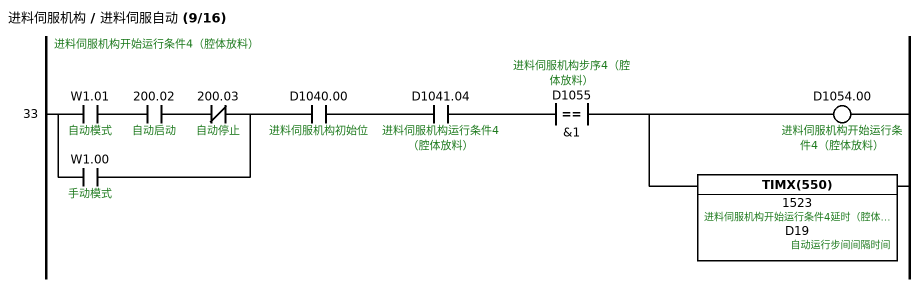
; [picture p120: 进料伺服机构 / 进料伺服自动, rungs 33-33]
; rung 33: 进料伺服机构开始运行条件4（腔体放料）
LD W1.01  ; 自动模式
AND 200.02  ; 自动启动
ANDNOT 200.03  ; 自动停止
OR W1.00  ; 手动模式
AND D1040.00  ; 进料伺服机构初始位
AND D1041.04  ; 进料伺服机构运行条件4（腔体放料）
AND=(300) D1055 &1  ; 进料伺服机构步序4（腔体放料）
OUT D1054.00  ; 进料伺服机构开始运行条件4（腔体放料）
TIMX(550) 1523 D19  ; 自动运行步间间隔时间, 进料伺服机构开始运行条件4延时（腔体放料）

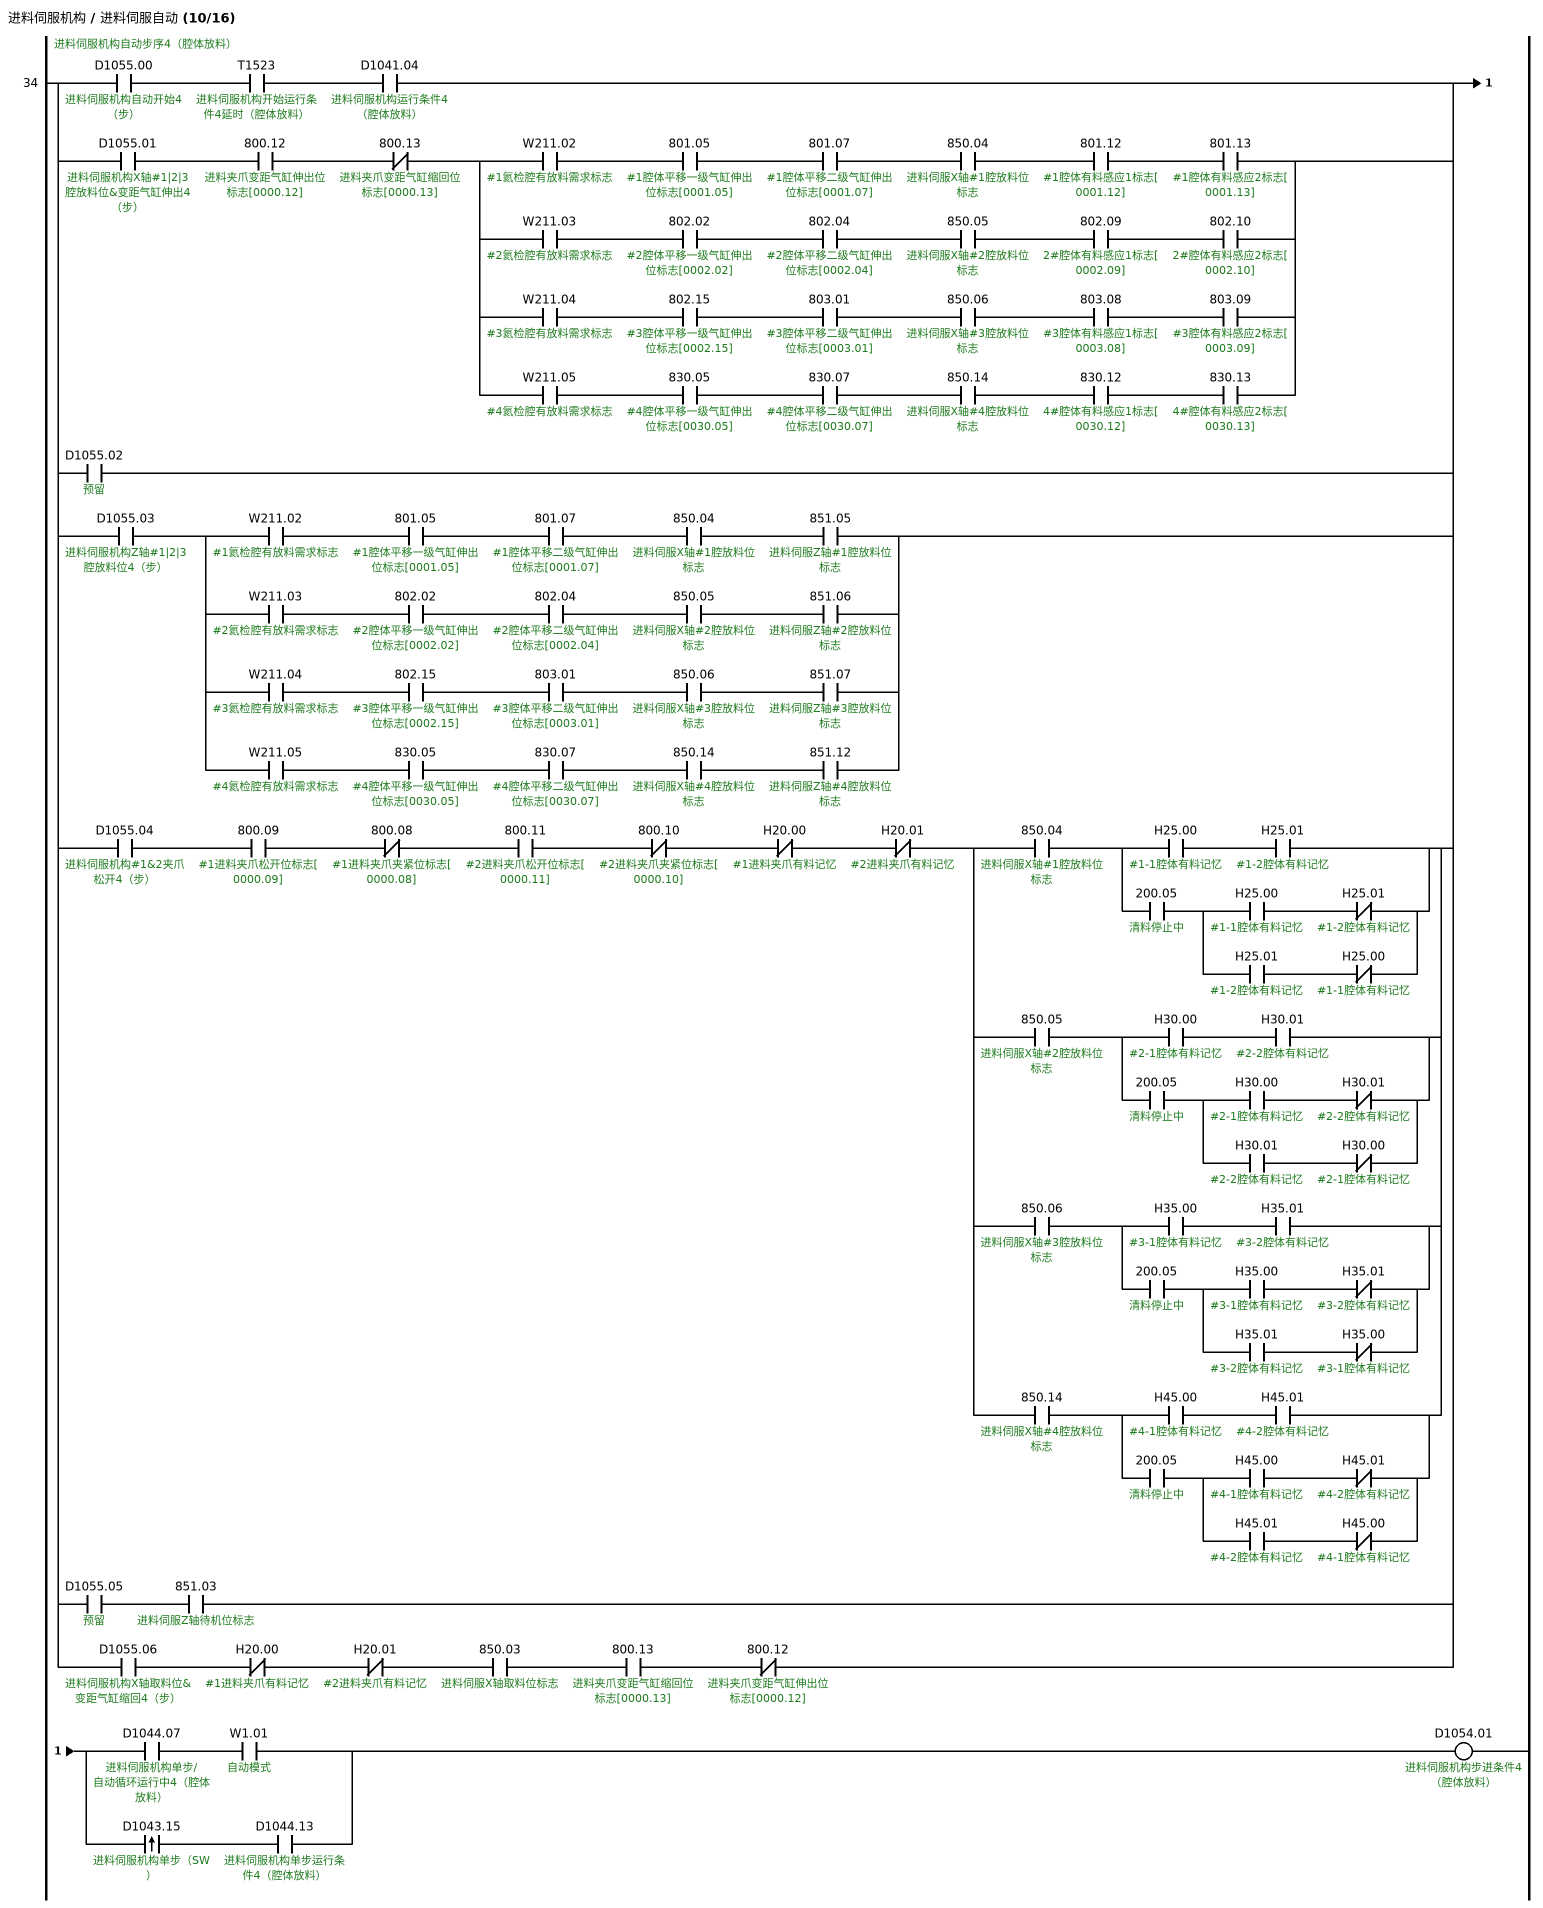
; rung 34: 进料伺服机构自动步序4（腔体放料）
LD D1055.00  ; 进料伺服机构自动开始4（步）
AND T1523  ; 进料伺服机构开始运行条件4延时（腔体放料）
AND D1041.04  ; 进料伺服机构运行条件4（腔体放料）
LD D1055.01  ; 进料伺服机构X轴#1|2|3腔放料位&变距气缸伸出4（步）
AND 800.12  ; 进料夹爪变距气缸伸出位标志[0000.12]
ANDNOT 800.13  ; 进料夹爪变距气缸缩回位标志[0000.13]
LD W211.02  ; #1氦检腔有放料需求标志
AND 801.05  ; #1腔体平移一级气缸伸出位标志[0001.05]
AND 801.07  ; #1腔体平移二级气缸伸出位标志[0001.07]
AND 850.04  ; 进料伺服X轴#1腔放料位标志
AND 801.12  ; #1腔体有料感应1标志[0001.12]
AND 801.13  ; #1腔体有料感应2标志[0001.13]
LD W211.03  ; #2氦检腔有放料需求标志
AND 802.02  ; #2腔体平移一级气缸伸出位标志[0002.02]
AND 802.04  ; #2腔体平移二级气缸伸出位标志[0002.04]
AND 850.05  ; 进料伺服X轴#2腔放料位标志
AND 802.09  ; 2#腔体有料感应1标志[0002.09]
AND 802.10  ; 2#腔体有料感应2标志[0002.10]
ORLD
LD W211.04  ; #3氦检腔有放料需求标志
AND 802.15  ; #3腔体平移一级气缸伸出位标志[0002.15]
AND 803.01  ; #3腔体平移二级气缸伸出位标志[0003.01]
AND 850.06  ; 进料伺服X轴#3腔放料位标志
AND 803.08  ; #3腔体有料感应1标志[0003.08]
AND 803.09  ; #3腔体有料感应2标志[0003.09]
ORLD
LD W211.05  ; #4氦检腔有放料需求标志
AND 830.05  ; #4腔体平移一级气缸伸出位标志[0030.05]
AND 830.07  ; #4腔体平移二级气缸伸出位标志[0030.07]
AND 850.14  ; 进料伺服X轴#4腔放料位标志
AND 830.12  ; 4#腔体有料感应1标志[0030.12]
AND 830.13  ; 4#腔体有料感应2标志[0030.13]
ORLD
ANDLD
ORLD
OR D1055.02  ; 预留
LD D1055.03  ; 进料伺服机构Z轴#1|2|3腔放料位4（步）
LD W211.02  ; #1氦检腔有放料需求标志
AND 801.05  ; #1腔体平移一级气缸伸出位标志[0001.05]
AND 801.07  ; #1腔体平移二级气缸伸出位标志[0001.07]
AND 850.04  ; 进料伺服X轴#1腔放料位标志
AND 851.05  ; 进料伺服Z轴#1腔放料位标志
LD W211.03  ; #2氦检腔有放料需求标志
AND 802.02  ; #2腔体平移一级气缸伸出位标志[0002.02]
AND 802.04  ; #2腔体平移二级气缸伸出位标志[0002.04]
AND 850.05  ; 进料伺服X轴#2腔放料位标志
AND 851.06  ; 进料伺服Z轴#2腔放料位标志
ORLD
LD W211.04  ; #3氦检腔有放料需求标志
AND 802.15  ; #3腔体平移一级气缸伸出位标志[0002.15]
AND 803.01  ; #3腔体平移二级气缸伸出位标志[0003.01]
AND 850.06  ; 进料伺服X轴#3腔放料位标志
AND 851.07  ; 进料伺服Z轴#3腔放料位标志
ORLD
LD W211.05  ; #4氦检腔有放料需求标志
AND 830.05  ; #4腔体平移一级气缸伸出位标志[0030.05]
AND 830.07  ; #4腔体平移二级气缸伸出位标志[0030.07]
AND 850.14  ; 进料伺服X轴#4腔放料位标志
AND 851.12  ; 进料伺服Z轴#4腔放料位标志
ORLD
ANDLD
ORLD
LD D1055.04  ; 进料伺服机构#1&2夹爪松开4（步）
AND 800.09  ; #1进料夹爪松开位标志[0000.09]
ANDNOT 800.08  ; #1进料夹爪夹紧位标志[0000.08]
AND 800.11  ; #2进料夹爪松开位标志[0000.11]
ANDNOT 800.10  ; #2进料夹爪夹紧位标志[0000.10]
ANDNOT H20.00  ; #1进料夹爪有料记忆
ANDNOT H20.01  ; #2进料夹爪有料记忆
LD 850.04  ; 进料伺服X轴#1腔放料位标志
LD H25.00  ; #1-1腔体有料记忆
AND H25.01  ; #1-2腔体有料记忆
LD 200.05  ; 清料停止中
LD H25.00  ; #1-1腔体有料记忆
ANDNOT H25.01  ; #1-2腔体有料记忆
LD H25.01  ; #1-2腔体有料记忆
ANDNOT H25.00  ; #1-1腔体有料记忆
ORLD
ANDLD
ORLD
ANDLD
LD 850.05  ; 进料伺服X轴#2腔放料位标志
LD H30.00  ; #2-1腔体有料记忆
AND H30.01  ; #2-2腔体有料记忆
LD 200.05  ; 清料停止中
LD H30.00  ; #2-1腔体有料记忆
ANDNOT H30.01  ; #2-2腔体有料记忆
LD H30.01  ; #2-2腔体有料记忆
ANDNOT H30.00  ; #2-1腔体有料记忆
ORLD
ANDLD
ORLD
ANDLD
ORLD
LD 850.06  ; 进料伺服X轴#3腔放料位标志
LD H35.00  ; #3-1腔体有料记忆
AND H35.01  ; #3-2腔体有料记忆
LD 200.05  ; 清料停止中
LD H35.00  ; #3-1腔体有料记忆
ANDNOT H35.01  ; #3-2腔体有料记忆
LD H35.01  ; #3-2腔体有料记忆
ANDNOT H35.00  ; #3-1腔体有料记忆
ORLD
ANDLD
ORLD
ANDLD
ORLD
LD 850.14  ; 进料伺服X轴#4腔放料位标志
LD H45.00  ; #4-1腔体有料记忆
AND H45.01  ; #4-2腔体有料记忆
LD 200.05  ; 清料停止中
LD H45.00  ; #4-1腔体有料记忆
ANDNOT H45.01  ; #4-2腔体有料记忆
LD H45.01  ; #4-2腔体有料记忆
ANDNOT H45.00  ; #4-1腔体有料记忆
ORLD
ANDLD
ORLD
ANDLD
ORLD
ANDLD
ORLD
LD D1055.05  ; 预留
AND 851.03  ; 进料伺服Z轴待机位标志
ORLD
LD D1055.06  ; 进料伺服机构X轴取料位&变距气缸缩回4（步）
ANDNOT H20.00  ; #1进料夹爪有料记忆
ANDNOT H20.01  ; #2进料夹爪有料记忆
AND 850.03  ; 进料伺服X轴取料位标志
AND 800.13  ; 进料夹爪变距气缸缩回位标志[0000.13]
ANDNOT 800.12  ; 进料夹爪变距气缸伸出位标志[0000.12]
ORLD
LD D1044.07  ; 进料伺服机构单步/自动循环运行中4（腔体放料）
AND W1.01  ; 自动模式
@LD D1043.15  ; 进料伺服机构单步（SW）
AND D1044.13  ; 进料伺服机构单步运行条件4（腔体放料）
ORLD
ANDLD
OUT D1054.01  ; 进料伺服机构步进条件4（腔体放料）

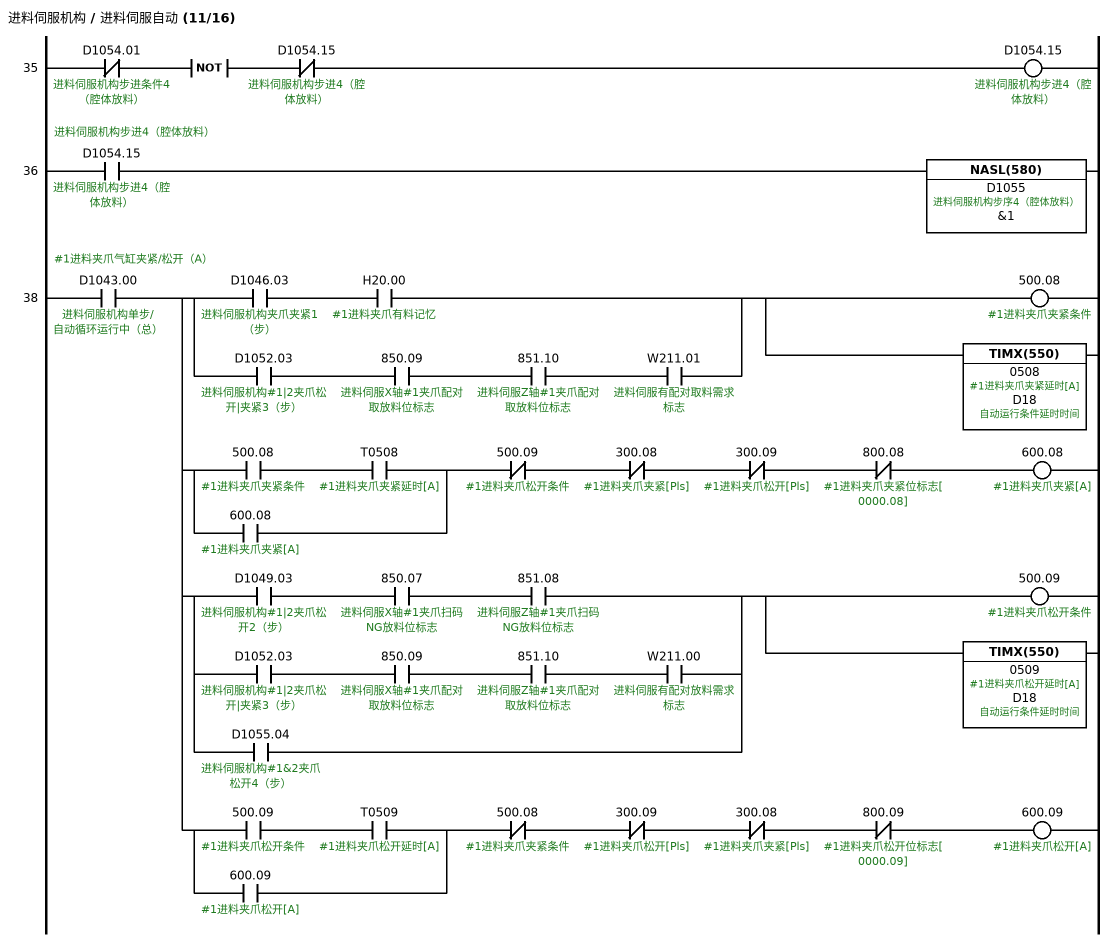
; rung 35
LDNOT D1054.01  ; 进料伺服机构步进条件4（腔体放料）
NOT(520)
ANDNOT D1054.15  ; 进料伺服机构步进4（腔体放料）
OUT D1054.15  ; 进料伺服机构步进4（腔体放料）
; rung 36: 进料伺服机构步进4（腔体放料）
LD D1054.15  ; 进料伺服机构步进4（腔体放料）
NASL(580) D1055 &1  ; 进料伺服机构步序4（腔体放料）
; rung 37: 进料伺服机构步序跳转程序4（腔体放料）
; rung 38: #1进料夹爪气缸夹紧/松开（A）
LD D1043.00  ; 进料伺服机构单步/自动循环运行中（总）
OUT TR0
LD D1046.03  ; 进料伺服机构夹爪夹紧1（步）
AND H20.00  ; #1进料夹爪有料记忆
LD D1052.03  ; 进料伺服机构#1|2夹爪松开|夹紧3（步）
AND 850.09  ; 进料伺服X轴#1夹爪配对取放料位标志
AND 851.10  ; 进料伺服Z轴#1夹爪配对取放料位标志
AND W211.01  ; 进料伺服有配对取料需求标志
ORLD
ANDLD
OUT 500.08  ; #1进料夹爪夹紧条件
TIMX(550) 0508 D18  ; 自动运行条件延时时间, #1进料夹爪夹紧延时[A]
LD TR0
LD 500.08  ; #1进料夹爪夹紧条件
AND T0508  ; #1进料夹爪夹紧延时[A]
OR 600.08  ; #1进料夹爪夹紧[A]
ANDLD
ANDNOT 500.09  ; #1进料夹爪松开条件
ANDNOT 300.08  ; #1进料夹爪夹紧[Pls]
ANDNOT 300.09  ; #1进料夹爪松开[Pls]
ANDNOT 800.08  ; #1进料夹爪夹紧位标志[0000.08]
OUT 600.08  ; #1进料夹爪夹紧[A]
LD TR0
LD D1049.03  ; 进料伺服机构#1|2夹爪松开2（步）
AND 850.07  ; 进料伺服X轴#1夹爪扫码NG放料位标志
AND 851.08  ; 进料伺服Z轴#1夹爪扫码NG放料位标志
LD D1052.03  ; 进料伺服机构#1|2夹爪松开|夹紧3（步）
AND 850.09  ; 进料伺服X轴#1夹爪配对取放料位标志
AND 851.10  ; 进料伺服Z轴#1夹爪配对取放料位标志
AND W211.00  ; 进料伺服有配对放料需求标志
ORLD
OR D1055.04  ; 进料伺服机构#1&2夹爪松开4（步）
ANDLD
OUT 500.09  ; #1进料夹爪松开条件
TIMX(550) 0509 D18  ; 自动运行条件延时时间, #1进料夹爪松开延时[A]
LD TR0
LD 500.09  ; #1进料夹爪松开条件
AND T0509  ; #1进料夹爪松开延时[A]
OR 600.09  ; #1进料夹爪松开[A]
ANDLD
ANDNOT 500.08  ; #1进料夹爪夹紧条件
ANDNOT 300.09  ; #1进料夹爪松开[Pls]
ANDNOT 300.08  ; #1进料夹爪夹紧[Pls]
ANDNOT 800.09  ; #1进料夹爪松开位标志[0000.09]
OUT 600.09  ; #1进料夹爪松开[A]

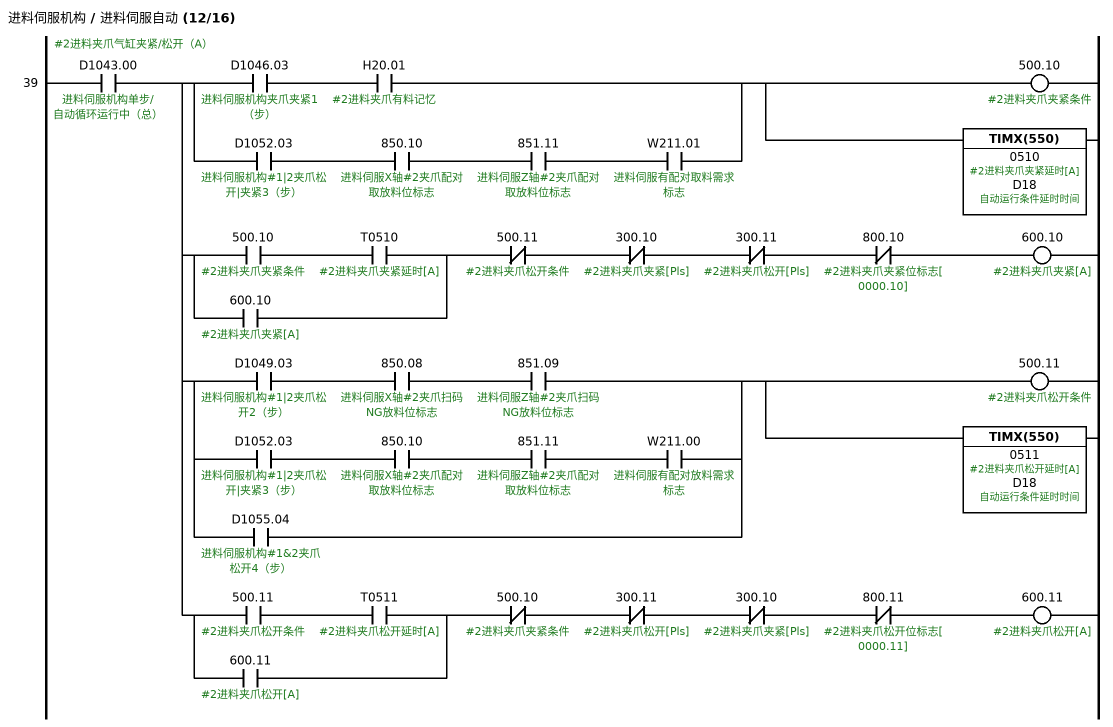
; rung 39: #2进料夹爪气缸夹紧/松开（A）
LD D1043.00  ; 进料伺服机构单步/自动循环运行中（总）
OUT TR0
LD D1046.03  ; 进料伺服机构夹爪夹紧1（步）
AND H20.01  ; #2进料夹爪有料记忆
LD D1052.03  ; 进料伺服机构#1|2夹爪松开|夹紧3（步）
AND 850.10  ; 进料伺服X轴#2夹爪配对取放料位标志
AND 851.11  ; 进料伺服Z轴#2夹爪配对取放料位标志
AND W211.01  ; 进料伺服有配对取料需求标志
ORLD
ANDLD
OUT 500.10  ; #2进料夹爪夹紧条件
TIMX(550) 0510 D18  ; 自动运行条件延时时间, #2进料夹爪夹紧延时[A]
LD TR0
LD 500.10  ; #2进料夹爪夹紧条件
AND T0510  ; #2进料夹爪夹紧延时[A]
OR 600.10  ; #2进料夹爪夹紧[A]
ANDLD
ANDNOT 500.11  ; #2进料夹爪松开条件
ANDNOT 300.10  ; #2进料夹爪夹紧[Pls]
ANDNOT 300.11  ; #2进料夹爪松开[Pls]
ANDNOT 800.10  ; #2进料夹爪夹紧位标志[0000.10]
OUT 600.10  ; #2进料夹爪夹紧[A]
LD TR0
LD D1049.03  ; 进料伺服机构#1|2夹爪松开2（步）
AND 850.08  ; 进料伺服X轴#2夹爪扫码NG放料位标志
AND 851.09  ; 进料伺服Z轴#2夹爪扫码NG放料位标志
LD D1052.03  ; 进料伺服机构#1|2夹爪松开|夹紧3（步）
AND 850.10  ; 进料伺服X轴#2夹爪配对取放料位标志
AND 851.11  ; 进料伺服Z轴#2夹爪配对取放料位标志
AND W211.00  ; 进料伺服有配对放料需求标志
ORLD
OR D1055.04  ; 进料伺服机构#1&2夹爪松开4（步）
ANDLD
OUT 500.11  ; #2进料夹爪松开条件
TIMX(550) 0511 D18  ; 自动运行条件延时时间, #2进料夹爪松开延时[A]
LD TR0
LD 500.11  ; #2进料夹爪松开条件
AND T0511  ; #2进料夹爪松开延时[A]
OR 600.11  ; #2进料夹爪松开[A]
ANDLD
ANDNOT 500.10  ; #2进料夹爪夹紧条件
ANDNOT 300.11  ; #2进料夹爪松开[Pls]
ANDNOT 300.10  ; #2进料夹爪夹紧[Pls]
ANDNOT 800.11  ; #2进料夹爪松开位标志[0000.11]
OUT 600.11  ; #2进料夹爪松开[A]

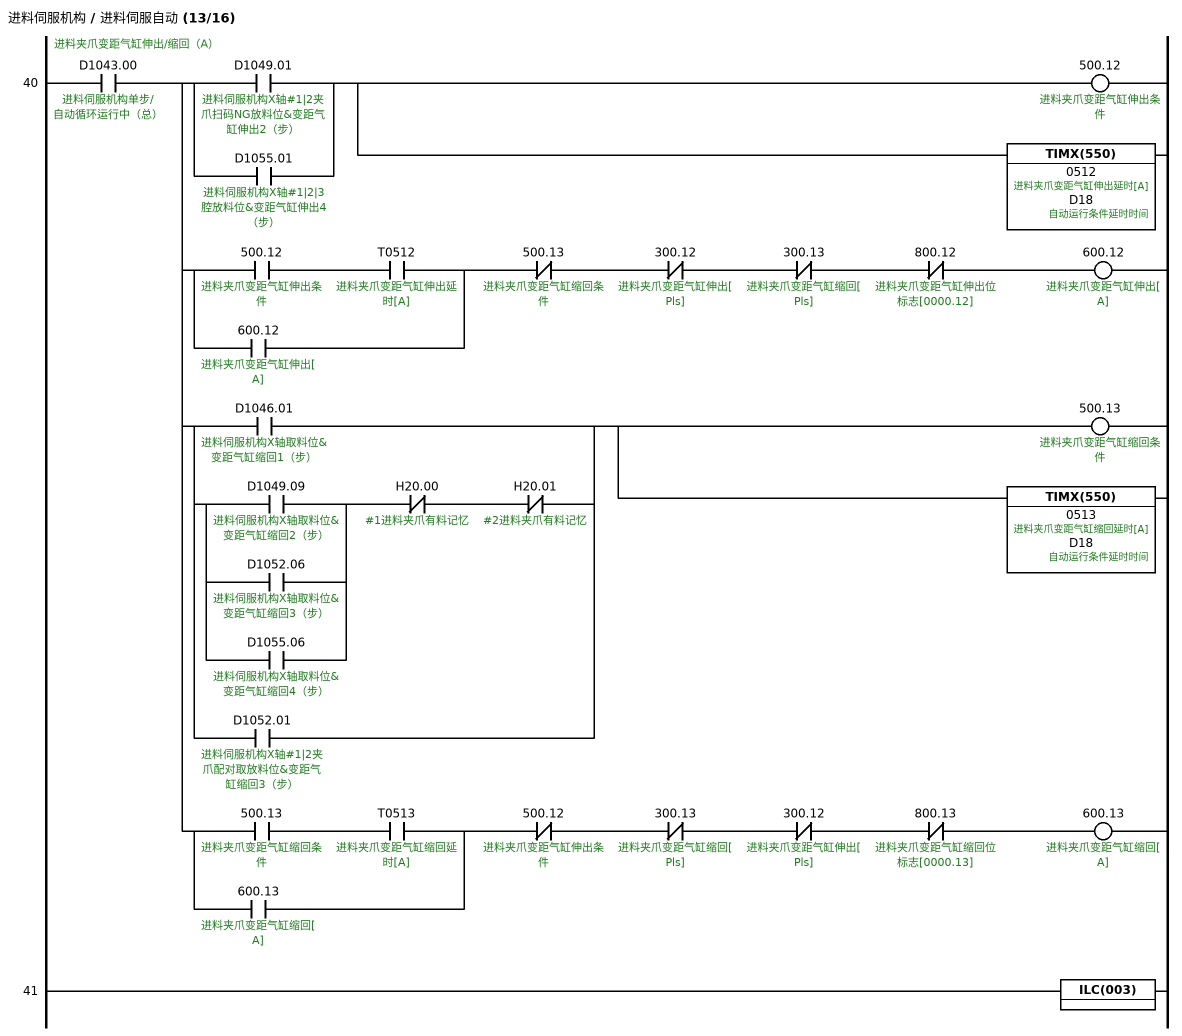
; rung 40: 进料夹爪变距气缸伸出/缩回（A）
LD D1043.00  ; 进料伺服机构单步/自动循环运行中（总）
OUT TR0
LD D1049.01  ; 进料伺服机构X轴#1|2夹爪扫码NG放料位&变距气缸伸出2（步）
OR D1055.01  ; 进料伺服机构X轴#1|2|3腔放料位&变距气缸伸出4（步）
ANDLD
OUT 500.12  ; 进料夹爪变距气缸伸出条件
TIMX(550) 0512 D18  ; 自动运行条件延时时间, 进料夹爪变距气缸伸出延时[A]
LD TR0
LD 500.12  ; 进料夹爪变距气缸伸出条件
AND T0512  ; 进料夹爪变距气缸伸出延时[A]
OR 600.12  ; 进料夹爪变距气缸伸出[A]
ANDLD
ANDNOT 500.13  ; 进料夹爪变距气缸缩回条件
ANDNOT 300.12  ; 进料夹爪变距气缸伸出[Pls]
ANDNOT 300.13  ; 进料夹爪变距气缸缩回[Pls]
ANDNOT 800.12  ; 进料夹爪变距气缸伸出位标志[0000.12]
OUT 600.12  ; 进料夹爪变距气缸伸出[A]
LD TR0
LD D1046.01  ; 进料伺服机构X轴取料位&变距气缸缩回1（步）
LD D1049.09  ; 进料伺服机构X轴取料位&变距气缸缩回2（步）
OR D1052.06  ; 进料伺服机构X轴取料位&变距气缸缩回3（步）
OR D1055.06  ; 进料伺服机构X轴取料位&变距气缸缩回4（步）
ANDNOT H20.00  ; #1进料夹爪有料记忆
ANDNOT H20.01  ; #2进料夹爪有料记忆
ORLD
OR D1052.01  ; 进料伺服机构X轴#1|2夹爪配对取放料位&变距气缸缩回3（步）
ANDLD
OUT 500.13  ; 进料夹爪变距气缸缩回条件
TIMX(550) 0513 D18  ; 自动运行条件延时时间, 进料夹爪变距气缸缩回延时[A]
LD TR0
LD 500.13  ; 进料夹爪变距气缸缩回条件
AND T0513  ; 进料夹爪变距气缸缩回延时[A]
OR 600.13  ; 进料夹爪变距气缸缩回[A]
ANDLD
ANDNOT 500.12  ; 进料夹爪变距气缸伸出条件
ANDNOT 300.13  ; 进料夹爪变距气缸缩回[Pls]
ANDNOT 300.12  ; 进料夹爪变距气缸伸出[Pls]
ANDNOT 800.13  ; 进料夹爪变距气缸缩回位标志[0000.13]
OUT 600.13  ; 进料夹爪变距气缸缩回[A]
; rung 41
ILC(003)

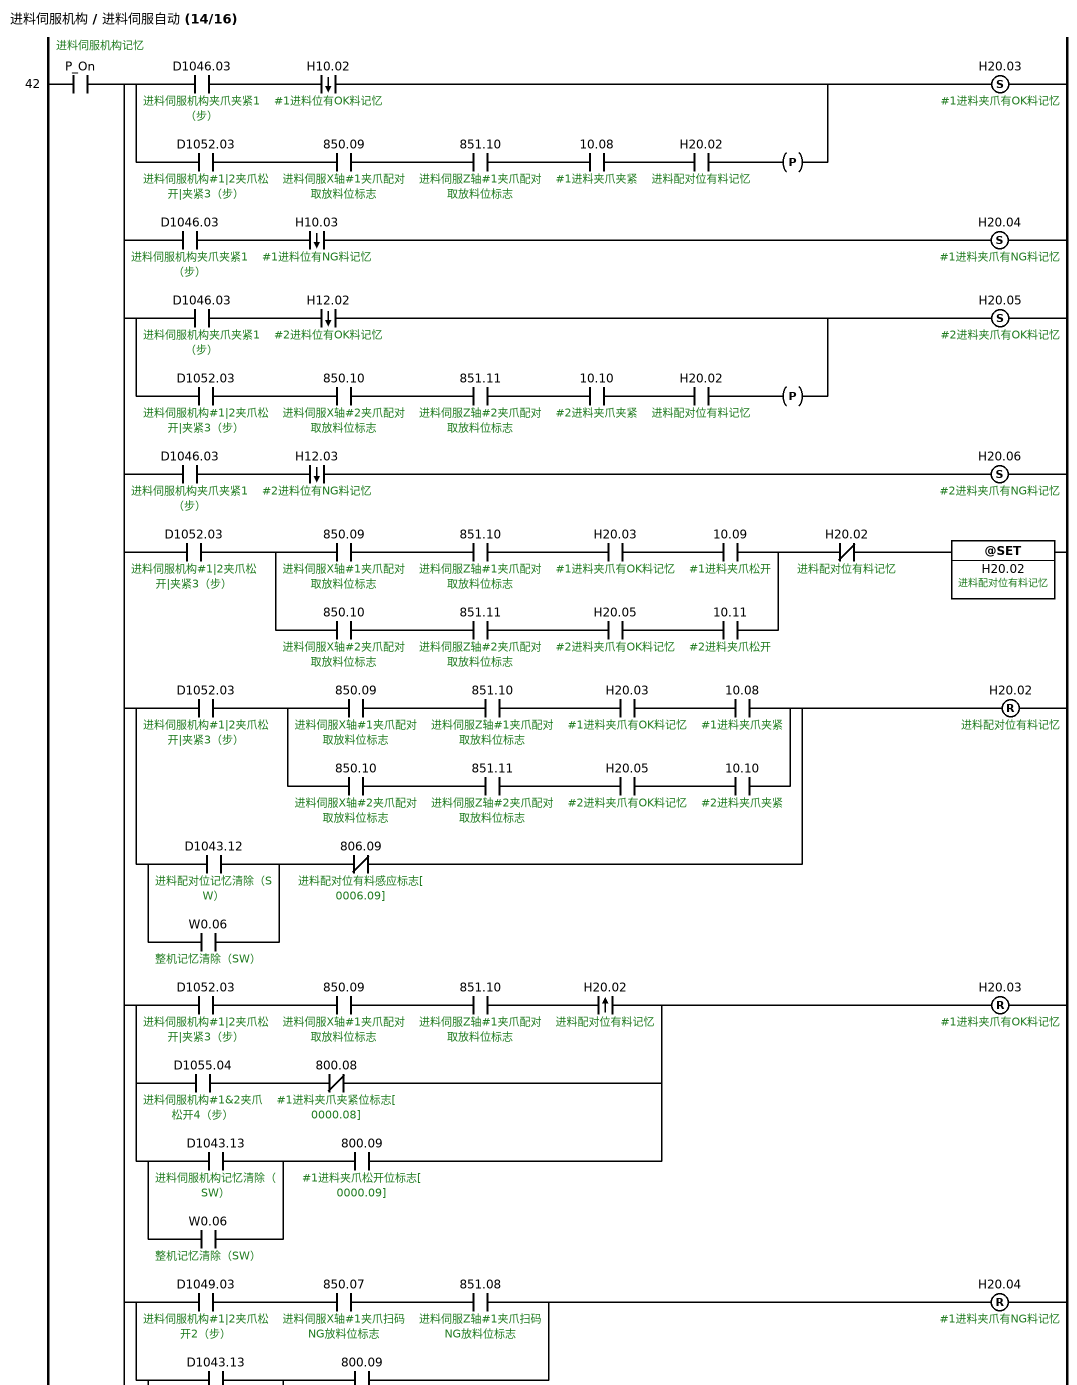

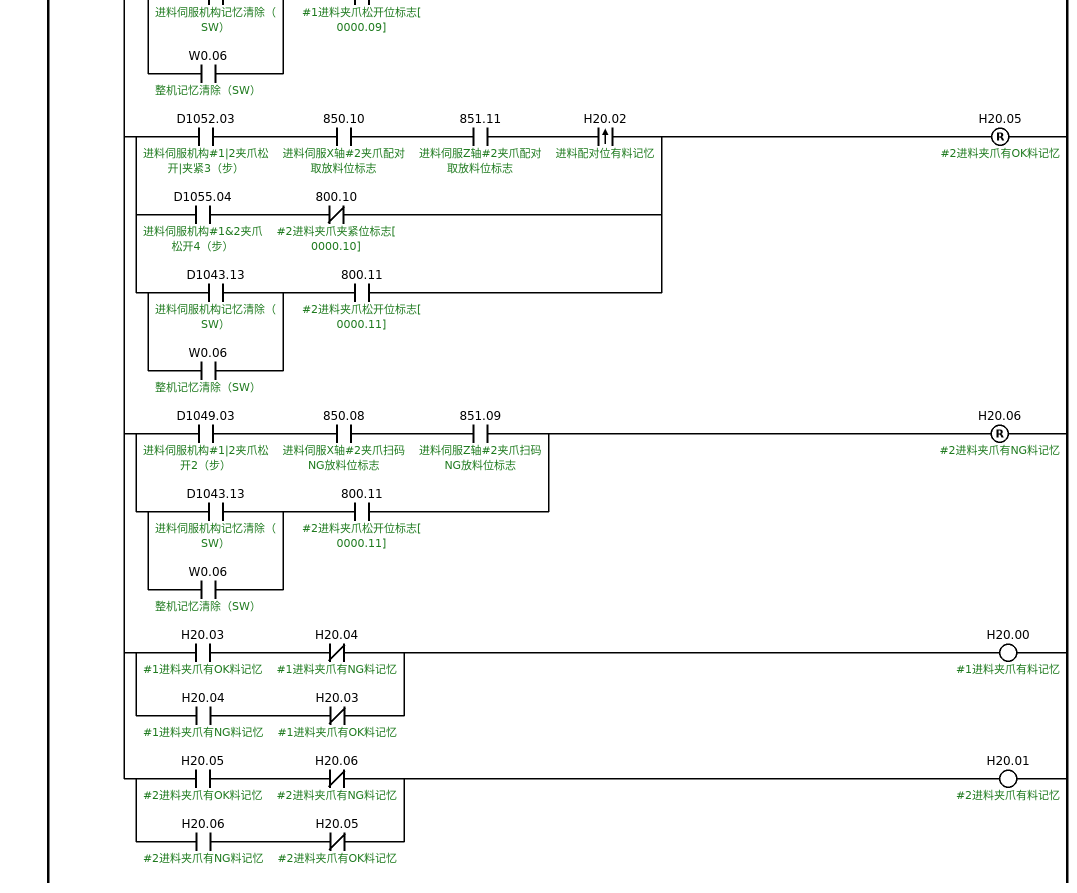
; rung 42: 进料伺服机构记忆
LD P_On
OUT TR0
LD D1046.03  ; 进料伺服机构夹爪夹紧1（步）
%AND H10.02  ; #1进料位有OK料记忆
LD D1052.03  ; 进料伺服机构#1|2夹爪松开|夹紧3（步）
AND 850.09  ; 进料伺服X轴#1夹爪配对取放料位标志
AND 851.10  ; 进料伺服Z轴#1夹爪配对取放料位标志
AND 10.08  ; #1进料夹爪夹紧
AND H20.02  ; 进料配对位有料记忆
UP(521)
ORLD
ANDLD
SET H20.03  ; #1进料夹爪有OK料记忆
LD TR0
AND D1046.03  ; 进料伺服机构夹爪夹紧1（步）
%AND H10.03  ; #1进料位有NG料记忆
SET H20.04  ; #1进料夹爪有NG料记忆
LD TR0
LD D1046.03  ; 进料伺服机构夹爪夹紧1（步）
%AND H12.02  ; #2进料位有OK料记忆
LD D1052.03  ; 进料伺服机构#1|2夹爪松开|夹紧3（步）
AND 850.10  ; 进料伺服X轴#2夹爪配对取放料位标志
AND 851.11  ; 进料伺服Z轴#2夹爪配对取放料位标志
AND 10.10  ; #2进料夹爪夹紧
AND H20.02  ; 进料配对位有料记忆
UP(521)
ORLD
ANDLD
SET H20.05  ; #2进料夹爪有OK料记忆
LD TR0
AND D1046.03  ; 进料伺服机构夹爪夹紧1（步）
%AND H12.03  ; #2进料位有NG料记忆
SET H20.06  ; #2进料夹爪有NG料记忆
LD TR0
AND D1052.03  ; 进料伺服机构#1|2夹爪松开|夹紧3（步）
LD 850.09  ; 进料伺服X轴#1夹爪配对取放料位标志
AND 851.10  ; 进料伺服Z轴#1夹爪配对取放料位标志
AND H20.03  ; #1进料夹爪有OK料记忆
AND 10.09  ; #1进料夹爪松开
LD 850.10  ; 进料伺服X轴#2夹爪配对取放料位标志
AND 851.11  ; 进料伺服Z轴#2夹爪配对取放料位标志
AND H20.05  ; #2进料夹爪有OK料记忆
AND 10.11  ; #2进料夹爪松开
ORLD
ANDLD
ANDNOT H20.02  ; 进料配对位有料记忆
@SET H20.02  ; 进料配对位有料记忆
LD TR0
LD D1052.03  ; 进料伺服机构#1|2夹爪松开|夹紧3（步）
LD 850.09  ; 进料伺服X轴#1夹爪配对取放料位标志
AND 851.10  ; 进料伺服Z轴#1夹爪配对取放料位标志
AND H20.03  ; #1进料夹爪有OK料记忆
AND 10.08  ; #1进料夹爪夹紧
LD 850.10  ; 进料伺服X轴#2夹爪配对取放料位标志
AND 851.11  ; 进料伺服Z轴#2夹爪配对取放料位标志
AND H20.05  ; #2进料夹爪有OK料记忆
AND 10.10  ; #2进料夹爪夹紧
ORLD
ANDLD
LD D1043.12  ; 进料配对位记忆清除（SW）
OR W0.06  ; 整机记忆清除（SW）
ANDNOT 806.09  ; 进料配对位有料感应标志[0006.09]
ORLD
ANDLD
RSET H20.02  ; 进料配对位有料记忆
LD TR0
LD D1052.03  ; 进料伺服机构#1|2夹爪松开|夹紧3（步）
AND 850.09  ; 进料伺服X轴#1夹爪配对取放料位标志
AND 851.10  ; 进料伺服Z轴#1夹爪配对取放料位标志
@AND H20.02  ; 进料配对位有料记忆
LD D1055.04  ; 进料伺服机构#1&2夹爪松开4（步）
ANDNOT 800.08  ; #1进料夹爪夹紧位标志[0000.08]
ORLD
LD D1043.13  ; 进料伺服机构记忆清除（SW）
OR W0.06  ; 整机记忆清除（SW）
AND 800.09  ; #1进料夹爪松开位标志[0000.09]
ORLD
ANDLD
RSET H20.03  ; #1进料夹爪有OK料记忆
LD TR0
LD D1049.03  ; 进料伺服机构#1|2夹爪松开2（步）
AND 850.07  ; 进料伺服X轴#1夹爪扫码NG放料位标志
AND 851.08  ; 进料伺服Z轴#1夹爪扫码NG放料位标志
LD D1043.13  ; 进料伺服机构记忆清除（SW）
OR W0.06  ; 整机记忆清除（SW）
AND 800.09  ; #1进料夹爪松开位标志[0000.09]
ORLD
ANDLD
RSET H20.04  ; #1进料夹爪有NG料记忆
LD TR0
LD D1052.03  ; 进料伺服机构#1|2夹爪松开|夹紧3（步）
AND 850.10  ; 进料伺服X轴#2夹爪配对取放料位标志
AND 851.11  ; 进料伺服Z轴#2夹爪配对取放料位标志
@AND H20.02  ; 进料配对位有料记忆
LD D1055.04  ; 进料伺服机构#1&2夹爪松开4（步）
ANDNOT 800.10  ; #2进料夹爪夹紧位标志[0000.10]
ORLD
LD D1043.13  ; 进料伺服机构记忆清除（SW）
OR W0.06  ; 整机记忆清除（SW）
AND 800.11  ; #2进料夹爪松开位标志[0000.11]
ORLD
ANDLD
RSET H20.05  ; #2进料夹爪有OK料记忆
LD TR0
LD D1049.03  ; 进料伺服机构#1|2夹爪松开2（步）
AND 850.08  ; 进料伺服X轴#2夹爪扫码NG放料位标志
AND 851.09  ; 进料伺服Z轴#2夹爪扫码NG放料位标志
LD D1043.13  ; 进料伺服机构记忆清除（SW）
OR W0.06  ; 整机记忆清除（SW）
AND 800.11  ; #2进料夹爪松开位标志[0000.11]
ORLD
ANDLD
RSET H20.06  ; #2进料夹爪有NG料记忆
LD TR0
LD H20.03  ; #1进料夹爪有OK料记忆
ANDNOT H20.04  ; #1进料夹爪有NG料记忆
LD H20.04  ; #1进料夹爪有NG料记忆
ANDNOT H20.03  ; #1进料夹爪有OK料记忆
ORLD
ANDLD
OUT H20.00  ; #1进料夹爪有料记忆
LD TR0
LD H20.05  ; #2进料夹爪有OK料记忆
ANDNOT H20.06  ; #2进料夹爪有NG料记忆
LD H20.06  ; #2进料夹爪有NG料记忆
ANDNOT H20.05  ; #2进料夹爪有OK料记忆
ORLD
ANDLD
OUT H20.01  ; #2进料夹爪有料记忆

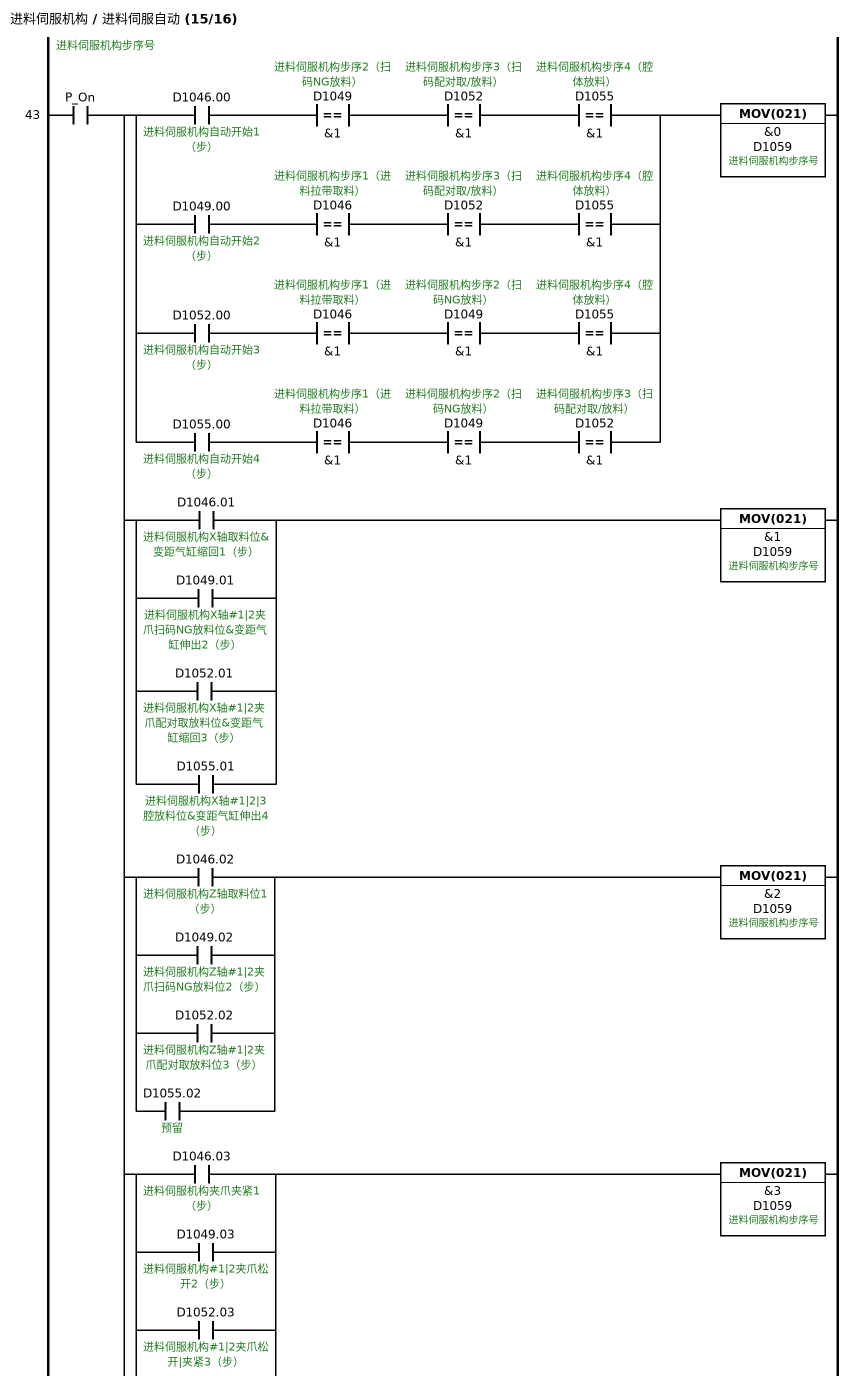

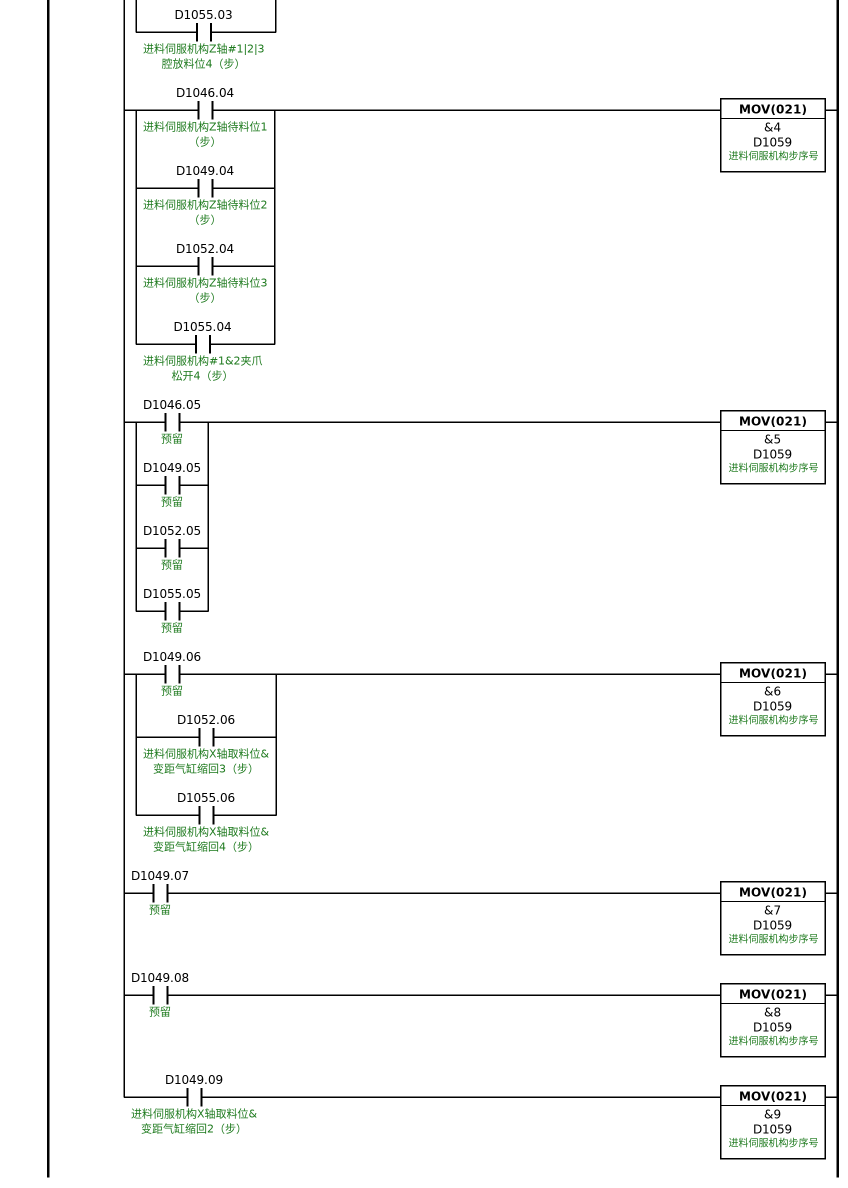
; rung 43: 进料伺服机构步序号
LD P_On
OUT TR0
LD D1046.00  ; 进料伺服机构自动开始1（步）
AND=(300) D1049 &1  ; 进料伺服机构步序2（扫码NG放料）
AND=(300) D1052 &1  ; 进料伺服机构步序3（扫码配对取/放料）
AND=(300) D1055 &1  ; 进料伺服机构步序4（腔体放料）
LD D1049.00  ; 进料伺服机构自动开始2（步）
AND=(300) D1046 &1  ; 进料伺服机构步序1（进料拉带取料）
AND=(300) D1052 &1  ; 进料伺服机构步序3（扫码配对取/放料）
AND=(300) D1055 &1  ; 进料伺服机构步序4（腔体放料）
ORLD
LD D1052.00  ; 进料伺服机构自动开始3（步）
AND=(300) D1046 &1  ; 进料伺服机构步序1（进料拉带取料）
AND=(300) D1049 &1  ; 进料伺服机构步序2（扫码NG放料）
AND=(300) D1055 &1  ; 进料伺服机构步序4（腔体放料）
ORLD
LD D1055.00  ; 进料伺服机构自动开始4（步）
AND=(300) D1046 &1  ; 进料伺服机构步序1（进料拉带取料）
AND=(300) D1049 &1  ; 进料伺服机构步序2（扫码NG放料）
AND=(300) D1052 &1  ; 进料伺服机构步序3（扫码配对取/放料）
ORLD
ANDLD
MOV(021) &0 D1059  ; 进料伺服机构步序号
LD TR0
LD D1046.01  ; 进料伺服机构X轴取料位&变距气缸缩回1（步）
OR D1049.01  ; 进料伺服机构X轴#1|2夹爪扫码NG放料位&变距气缸伸出2（步）
OR D1052.01  ; 进料伺服机构X轴#1|2夹爪配对取放料位&变距气缸缩回3（步）
OR D1055.01  ; 进料伺服机构X轴#1|2|3腔放料位&变距气缸伸出4（步）
ANDLD
MOV(021) &1 D1059  ; 进料伺服机构步序号
LD TR0
LD D1046.02  ; 进料伺服机构Z轴取料位1（步）
OR D1049.02  ; 进料伺服机构Z轴#1|2夹爪扫码NG放料位2（步）
OR D1052.02  ; 进料伺服机构Z轴#1|2夹爪配对取放料位3（步）
OR D1055.02  ; 预留
ANDLD
MOV(021) &2 D1059  ; 进料伺服机构步序号
LD TR0
LD D1046.03  ; 进料伺服机构夹爪夹紧1（步）
OR D1049.03  ; 进料伺服机构#1|2夹爪松开2（步）
OR D1052.03  ; 进料伺服机构#1|2夹爪松开|夹紧3（步）
OR D1055.03  ; 进料伺服机构Z轴#1|2|3腔放料位4（步）
ANDLD
MOV(021) &3 D1059  ; 进料伺服机构步序号
LD TR0
LD D1046.04  ; 进料伺服机构Z轴待料位1（步）
OR D1049.04  ; 进料伺服机构Z轴待料位2（步）
OR D1052.04  ; 进料伺服机构Z轴待料位3（步）
OR D1055.04  ; 进料伺服机构#1&2夹爪松开4（步）
ANDLD
MOV(021) &4 D1059  ; 进料伺服机构步序号
LD TR0
LD D1046.05  ; 预留
OR D1049.05  ; 预留
OR D1052.05  ; 预留
OR D1055.05  ; 预留
ANDLD
MOV(021) &5 D1059  ; 进料伺服机构步序号
LD TR0
LD D1049.06  ; 预留
OR D1052.06  ; 进料伺服机构X轴取料位&变距气缸缩回3（步）
OR D1055.06  ; 进料伺服机构X轴取料位&变距气缸缩回4（步）
ANDLD
MOV(021) &6 D1059  ; 进料伺服机构步序号
LD TR0
AND D1049.07  ; 预留
MOV(021) &7 D1059  ; 进料伺服机构步序号
LD TR0
AND D1049.08  ; 预留
MOV(021) &8 D1059  ; 进料伺服机构步序号
LD TR0
AND D1049.09  ; 进料伺服机构X轴取料位&变距气缸缩回2（步）
MOV(021) &9 D1059  ; 进料伺服机构步序号

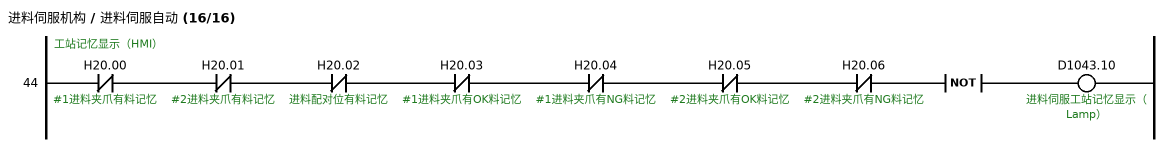
; rung 44: 工站记忆显示（HMI）
LDNOT H20.00  ; #1进料夹爪有料记忆
ANDNOT H20.01  ; #2进料夹爪有料记忆
ANDNOT H20.02  ; 进料配对位有料记忆
ANDNOT H20.03  ; #1进料夹爪有OK料记忆
ANDNOT H20.04  ; #1进料夹爪有NG料记忆
ANDNOT H20.05  ; #2进料夹爪有OK料记忆
ANDNOT H20.06  ; #2进料夹爪有NG料记忆
NOT(520)
OUT D1043.10  ; 进料伺服工站记忆显示（Lamp）

### Section 工站复位

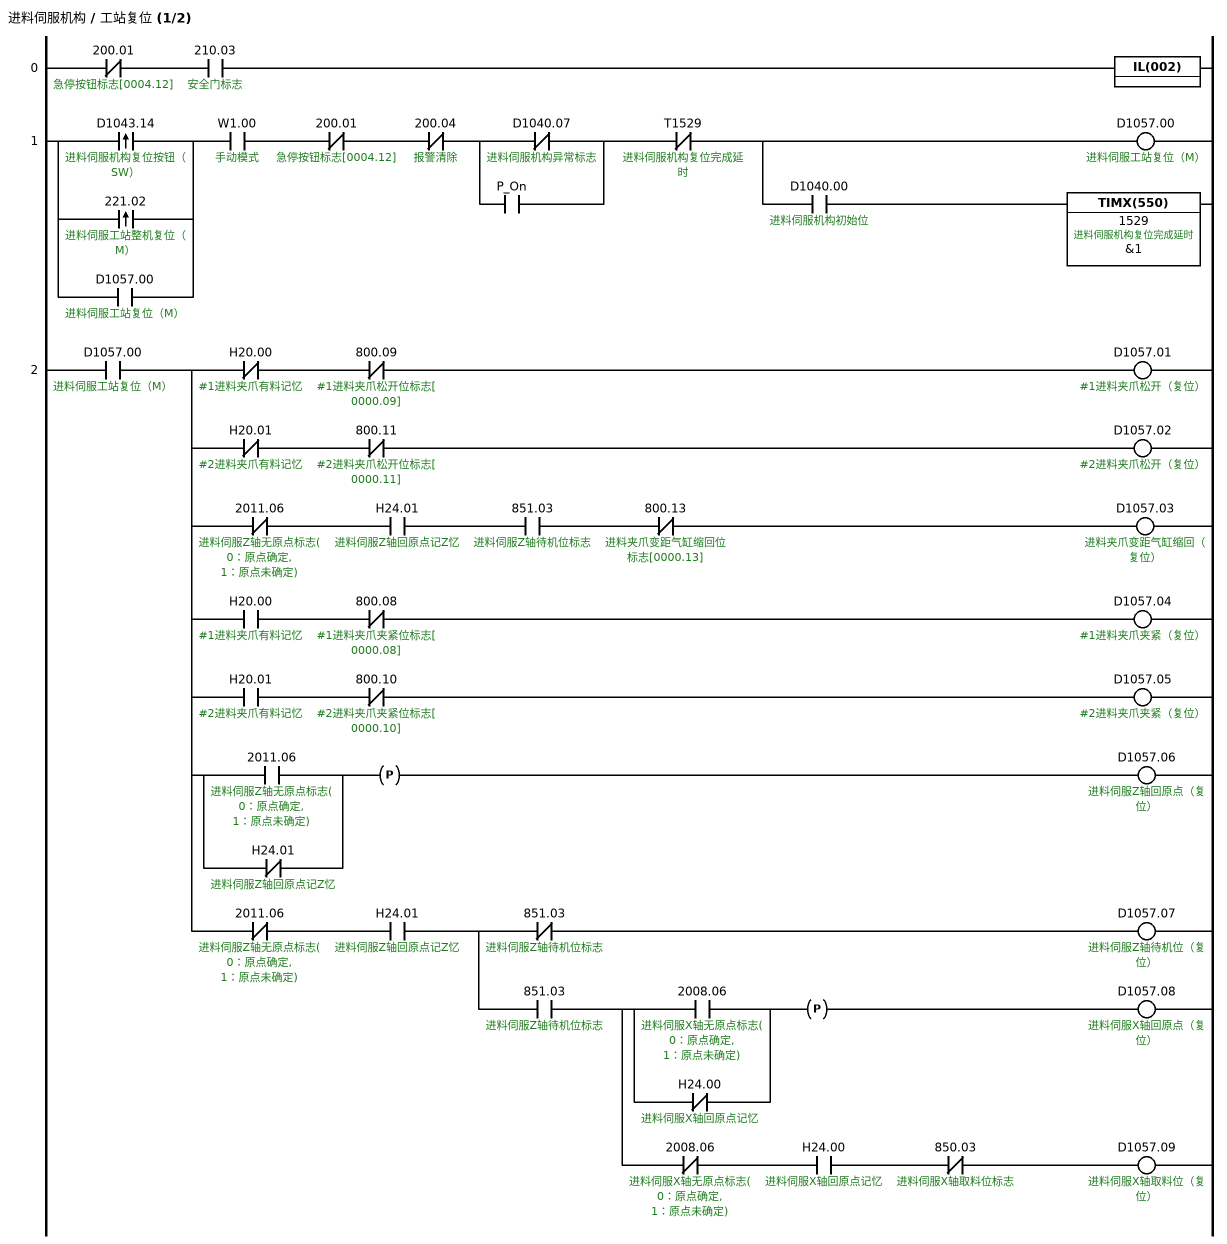
; rung 0
LDNOT 200.01  ; 急停按钮标志[0004.12]
AND 210.03  ; 安全门标志
IL(002)
; rung 1
@LD D1043.14  ; 进料伺服机构复位按钮（SW）
@OR 221.02  ; 进料伺服工站整机复位（M）
OR D1057.00  ; 进料伺服工站复位（M）
AND W1.00  ; 手动模式
ANDNOT 200.01  ; 急停按钮标志[0004.12]
ANDNOT 200.04  ; 报警清除
LDNOT D1040.07  ; 进料伺服机构异常标志
OR P_On
ANDLD
ANDNOT T1529  ; 进料伺服机构复位完成延时
OUT D1057.00  ; 进料伺服工站复位（M）
AND D1040.00  ; 进料伺服机构初始位
TIMX(550) 1529 &1  ; 进料伺服机构复位完成延时
; rung 2
LD D1057.00  ; 进料伺服工站复位（M）
OUT TR0
ANDNOT H20.00  ; #1进料夹爪有料记忆
ANDNOT 800.09  ; #1进料夹爪松开位标志[0000.09]
OUT D1057.01  ; #1进料夹爪松开（复位）
LD TR0
ANDNOT H20.01  ; #2进料夹爪有料记忆
ANDNOT 800.11  ; #2进料夹爪松开位标志[0000.11]
OUT D1057.02  ; #2进料夹爪松开（复位）
LD TR0
ANDNOT 2011.06  ; 进料伺服Z轴无原点标志(0：原点确定,1：原点未确定)
AND H24.01  ; 进料伺服Z轴回原点记Z忆
AND 851.03  ; 进料伺服Z轴待机位标志
ANDNOT 800.13  ; 进料夹爪变距气缸缩回位标志[0000.13]
OUT D1057.03  ; 进料夹爪变距气缸缩回（复位）
LD TR0
AND H20.00  ; #1进料夹爪有料记忆
ANDNOT 800.08  ; #1进料夹爪夹紧位标志[0000.08]
OUT D1057.04  ; #1进料夹爪夹紧（复位）
LD TR0
AND H20.01  ; #2进料夹爪有料记忆
ANDNOT 800.10  ; #2进料夹爪夹紧位标志[0000.10]
OUT D1057.05  ; #2进料夹爪夹紧（复位）
LD TR0
LD 2011.06  ; 进料伺服Z轴无原点标志(0：原点确定,1：原点未确定)
ORNOT H24.01  ; 进料伺服Z轴回原点记Z忆
ANDLD
UP(521)
OUT D1057.06  ; 进料伺服Z轴回原点（复位）
LD TR0
ANDNOT 2011.06  ; 进料伺服Z轴无原点标志(0：原点确定,1：原点未确定)
AND H24.01  ; 进料伺服Z轴回原点记Z忆
OUT TR0
ANDNOT 851.03  ; 进料伺服Z轴待机位标志
OUT D1057.07  ; 进料伺服Z轴待机位（复位）
LD TR0
AND 851.03  ; 进料伺服Z轴待机位标志
OUT TR0
LD 2008.06  ; 进料伺服X轴无原点标志(0：原点确定,1：原点未确定)
ORNOT H24.00  ; 进料伺服X轴回原点记忆
ANDLD
UP(521)
OUT D1057.08  ; 进料伺服X轴回原点（复位）
LD TR0
ANDNOT 2008.06  ; 进料伺服X轴无原点标志(0：原点确定,1：原点未确定)
AND H24.00  ; 进料伺服X轴回原点记忆
ANDNOT 850.03  ; 进料伺服X轴取料位标志
OUT D1057.09  ; 进料伺服X轴取料位（复位）

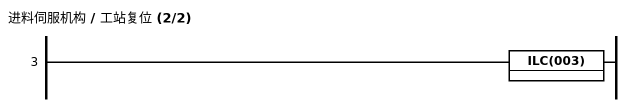
; rung 3
ILC(003)

### Section 指示灯

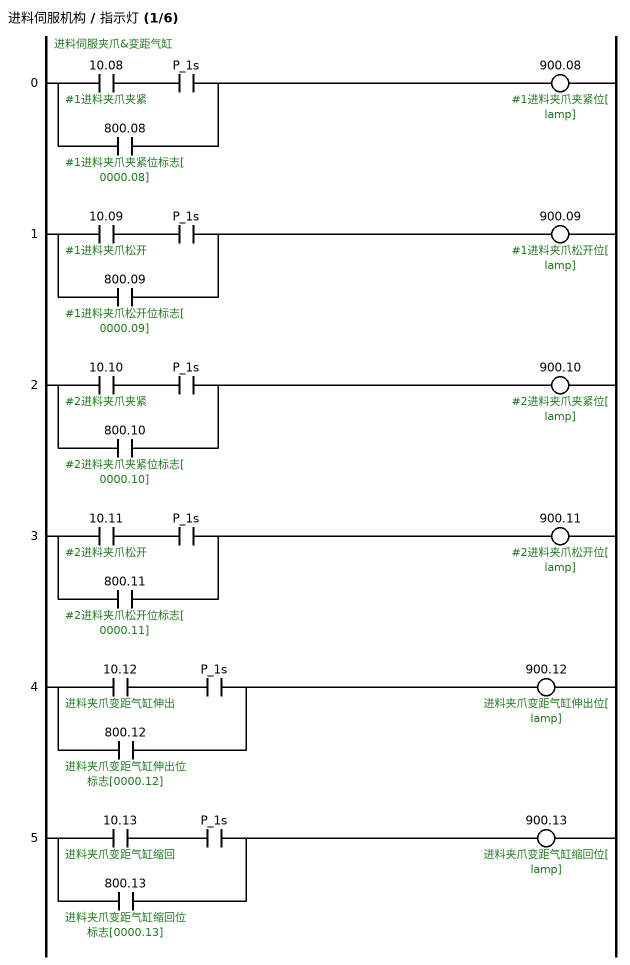
; rung 0: 进料伺服夹爪&变距气缸
LD 10.08  ; #1进料夹爪夹紧
AND P_1s
OR 800.08  ; #1进料夹爪夹紧位标志[0000.08]
OUT 900.08  ; #1进料夹爪夹紧位[lamp]
; rung 1
LD 10.09  ; #1进料夹爪松开
AND P_1s
OR 800.09  ; #1进料夹爪松开位标志[0000.09]
OUT 900.09  ; #1进料夹爪松开位[lamp]
; rung 2
LD 10.10  ; #2进料夹爪夹紧
AND P_1s
OR 800.10  ; #2进料夹爪夹紧位标志[0000.10]
OUT 900.10  ; #2进料夹爪夹紧位[lamp]
; rung 3
LD 10.11  ; #2进料夹爪松开
AND P_1s
OR 800.11  ; #2进料夹爪松开位标志[0000.11]
OUT 900.11  ; #2进料夹爪松开位[lamp]
; rung 4
LD 10.12  ; 进料夹爪变距气缸伸出
AND P_1s
OR 800.12  ; 进料夹爪变距气缸伸出位标志[0000.12]
OUT 900.12  ; 进料夹爪变距气缸伸出位[lamp]
; rung 5
LD 10.13  ; 进料夹爪变距气缸缩回
AND P_1s
OR 800.13  ; 进料夹爪变距气缸缩回位标志[0000.13]
OUT 900.13  ; 进料夹爪变距气缸缩回位[lamp]

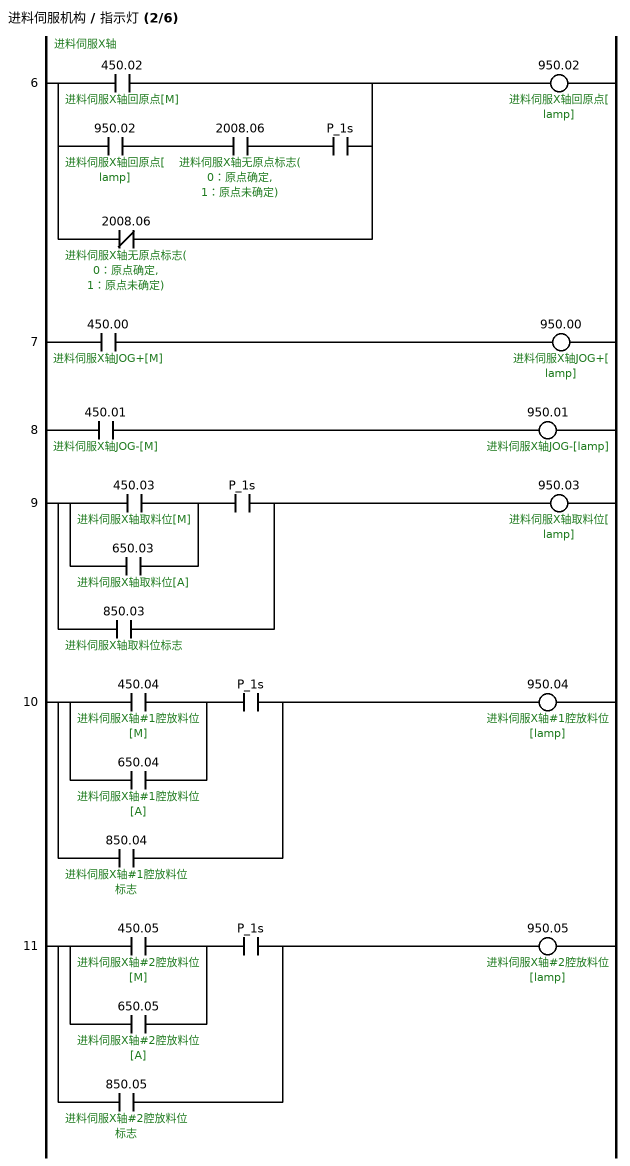
; rung 6: 进料伺服X轴
LD 450.02  ; 进料伺服X轴回原点[M]
LD 950.02  ; 进料伺服X轴回原点[lamp]
AND 2008.06  ; 进料伺服X轴无原点标志(0：原点确定,1：原点未确定)
AND P_1s
ORLD
ORNOT 2008.06  ; 进料伺服X轴无原点标志(0：原点确定,1：原点未确定)
OUT 950.02  ; 进料伺服X轴回原点[lamp]
; rung 7
LD 450.00  ; 进料伺服X轴JOG+[M]
OUT 950.00  ; 进料伺服X轴JOG+[lamp]
; rung 8
LD 450.01  ; 进料伺服X轴JOG-[M]
OUT 950.01  ; 进料伺服X轴JOG-[lamp]
; rung 9
LD 450.03  ; 进料伺服X轴取料位[M]
OR 650.03  ; 进料伺服X轴取料位[A]
AND P_1s
OR 850.03  ; 进料伺服X轴取料位标志
OUT 950.03  ; 进料伺服X轴取料位[lamp]
; rung 10
LD 450.04  ; 进料伺服X轴#1腔放料位[M]
OR 650.04  ; 进料伺服X轴#1腔放料位[A]
AND P_1s
OR 850.04  ; 进料伺服X轴#1腔放料位标志
OUT 950.04  ; 进料伺服X轴#1腔放料位[lamp]
; rung 11
LD 450.05  ; 进料伺服X轴#2腔放料位[M]
OR 650.05  ; 进料伺服X轴#2腔放料位[A]
AND P_1s
OR 850.05  ; 进料伺服X轴#2腔放料位标志
OUT 950.05  ; 进料伺服X轴#2腔放料位[lamp]

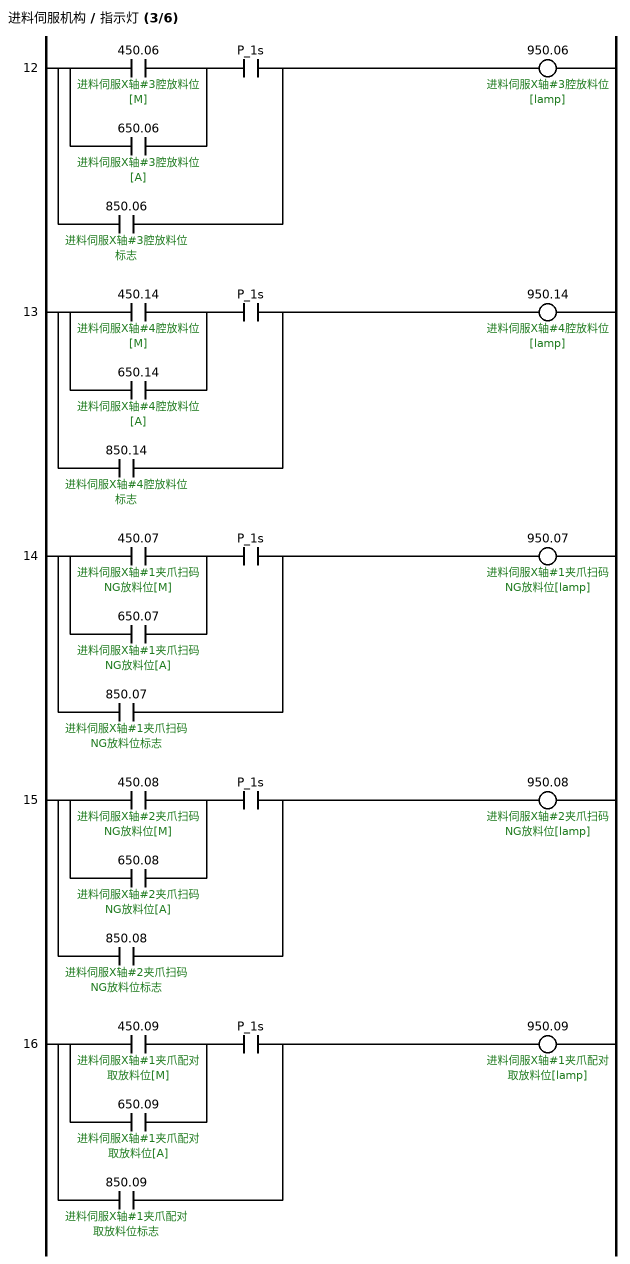
; rung 12
LD 450.06  ; 进料伺服X轴#3腔放料位[M]
OR 650.06  ; 进料伺服X轴#3腔放料位[A]
AND P_1s
OR 850.06  ; 进料伺服X轴#3腔放料位标志
OUT 950.06  ; 进料伺服X轴#3腔放料位[lamp]
; rung 13
LD 450.14  ; 进料伺服X轴#4腔放料位[M]
OR 650.14  ; 进料伺服X轴#4腔放料位[A]
AND P_1s
OR 850.14  ; 进料伺服X轴#4腔放料位标志
OUT 950.14  ; 进料伺服X轴#4腔放料位[lamp]
; rung 14
LD 450.07  ; 进料伺服X轴#1夹爪扫码NG放料位[M]
OR 650.07  ; 进料伺服X轴#1夹爪扫码NG放料位[A]
AND P_1s
OR 850.07  ; 进料伺服X轴#1夹爪扫码NG放料位标志
OUT 950.07  ; 进料伺服X轴#1夹爪扫码NG放料位[lamp]
; rung 15
LD 450.08  ; 进料伺服X轴#2夹爪扫码NG放料位[M]
OR 650.08  ; 进料伺服X轴#2夹爪扫码NG放料位[A]
AND P_1s
OR 850.08  ; 进料伺服X轴#2夹爪扫码NG放料位标志
OUT 950.08  ; 进料伺服X轴#2夹爪扫码NG放料位[lamp]
; rung 16
LD 450.09  ; 进料伺服X轴#1夹爪配对取放料位[M]
OR 650.09  ; 进料伺服X轴#1夹爪配对取放料位[A]
AND P_1s
OR 850.09  ; 进料伺服X轴#1夹爪配对取放料位标志
OUT 950.09  ; 进料伺服X轴#1夹爪配对取放料位[lamp]

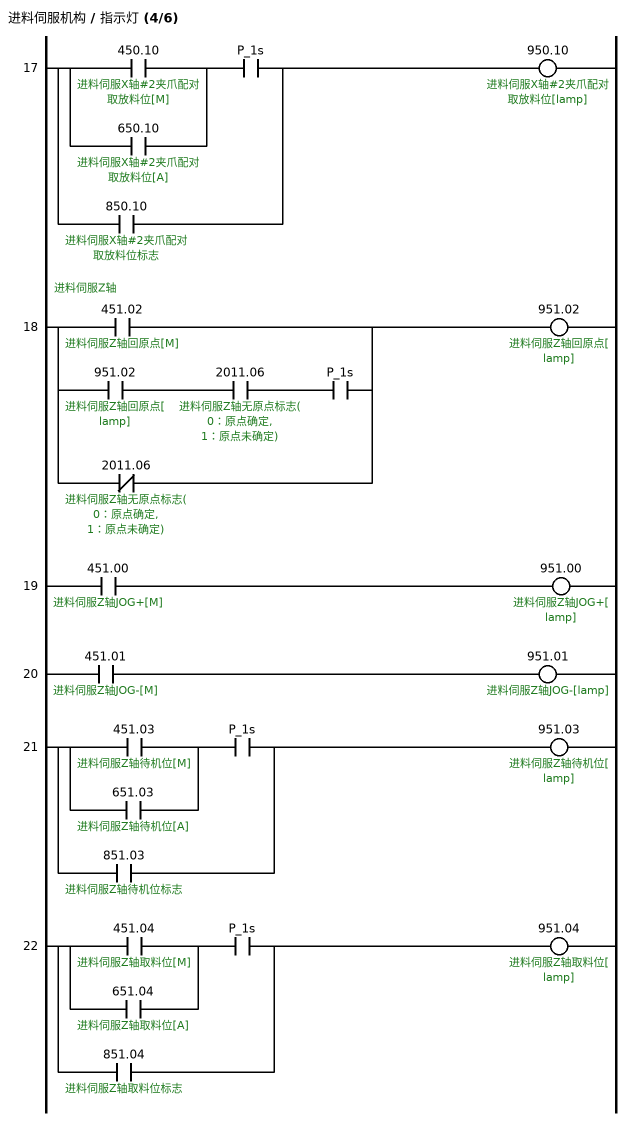
; rung 17
LD 450.10  ; 进料伺服X轴#2夹爪配对取放料位[M]
OR 650.10  ; 进料伺服X轴#2夹爪配对取放料位[A]
AND P_1s
OR 850.10  ; 进料伺服X轴#2夹爪配对取放料位标志
OUT 950.10  ; 进料伺服X轴#2夹爪配对取放料位[lamp]
; rung 18: 进料伺服Z轴
LD 451.02  ; 进料伺服Z轴回原点[M]
LD 951.02  ; 进料伺服Z轴回原点[lamp]
AND 2011.06  ; 进料伺服Z轴无原点标志(0：原点确定,1：原点未确定)
AND P_1s
ORLD
ORNOT 2011.06  ; 进料伺服Z轴无原点标志(0：原点确定,1：原点未确定)
OUT 951.02  ; 进料伺服Z轴回原点[lamp]
; rung 19
LD 451.00  ; 进料伺服Z轴JOG+[M]
OUT 951.00  ; 进料伺服Z轴JOG+[lamp]
; rung 20
LD 451.01  ; 进料伺服Z轴JOG-[M]
OUT 951.01  ; 进料伺服Z轴JOG-[lamp]
; rung 21
LD 451.03  ; 进料伺服Z轴待机位[M]
OR 651.03  ; 进料伺服Z轴待机位[A]
AND P_1s
OR 851.03  ; 进料伺服Z轴待机位标志
OUT 951.03  ; 进料伺服Z轴待机位[lamp]
; rung 22
LD 451.04  ; 进料伺服Z轴取料位[M]
OR 651.04  ; 进料伺服Z轴取料位[A]
AND P_1s
OR 851.04  ; 进料伺服Z轴取料位标志
OUT 951.04  ; 进料伺服Z轴取料位[lamp]

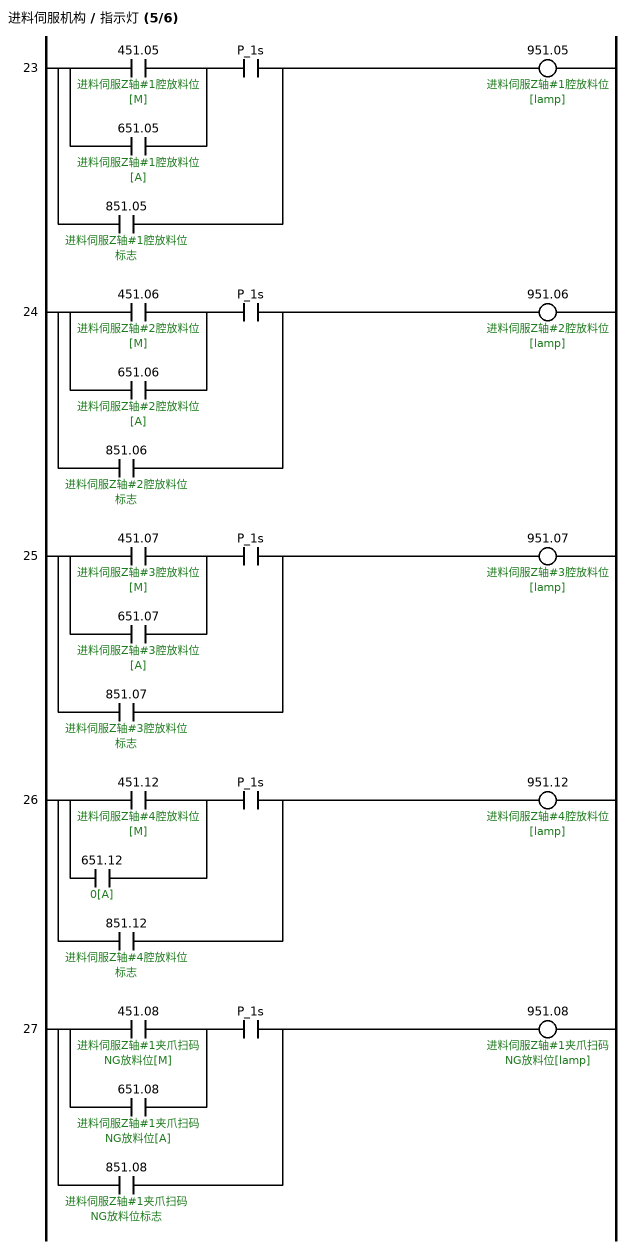
; rung 23
LD 451.05  ; 进料伺服Z轴#1腔放料位[M]
OR 651.05  ; 进料伺服Z轴#1腔放料位[A]
AND P_1s
OR 851.05  ; 进料伺服Z轴#1腔放料位标志
OUT 951.05  ; 进料伺服Z轴#1腔放料位[lamp]
; rung 24
LD 451.06  ; 进料伺服Z轴#2腔放料位[M]
OR 651.06  ; 进料伺服Z轴#2腔放料位[A]
AND P_1s
OR 851.06  ; 进料伺服Z轴#2腔放料位标志
OUT 951.06  ; 进料伺服Z轴#2腔放料位[lamp]
; rung 25
LD 451.07  ; 进料伺服Z轴#3腔放料位[M]
OR 651.07  ; 进料伺服Z轴#3腔放料位[A]
AND P_1s
OR 851.07  ; 进料伺服Z轴#3腔放料位标志
OUT 951.07  ; 进料伺服Z轴#3腔放料位[lamp]
; rung 26
LD 451.12  ; 进料伺服Z轴#4腔放料位[M]
OR 651.12  ; 0[A]
AND P_1s
OR 851.12  ; 进料伺服Z轴#4腔放料位标志
OUT 951.12  ; 进料伺服Z轴#4腔放料位[lamp]
; rung 27
LD 451.08  ; 进料伺服Z轴#1夹爪扫码NG放料位[M]
OR 651.08  ; 进料伺服Z轴#1夹爪扫码NG放料位[A]
AND P_1s
OR 851.08  ; 进料伺服Z轴#1夹爪扫码NG放料位标志
OUT 951.08  ; 进料伺服Z轴#1夹爪扫码NG放料位[lamp]

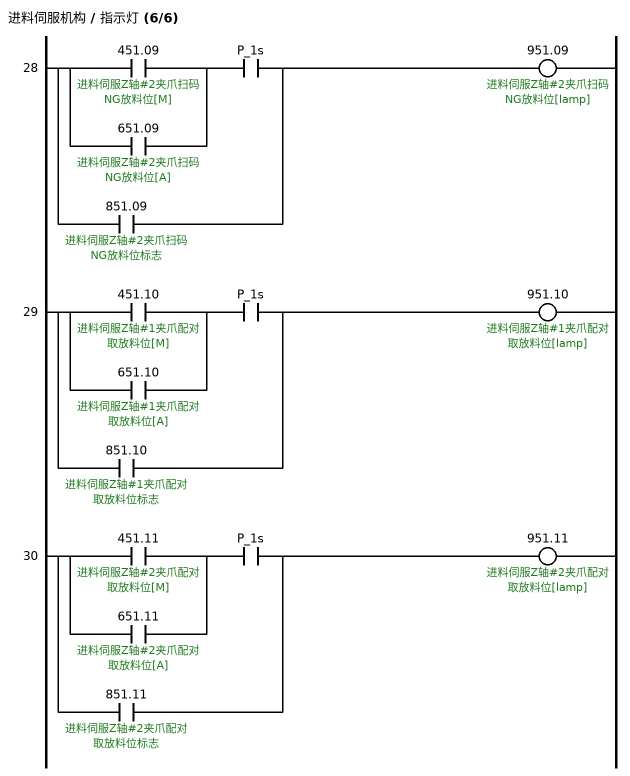
; rung 28
LD 451.09  ; 进料伺服Z轴#2夹爪扫码NG放料位[M]
OR 651.09  ; 进料伺服Z轴#2夹爪扫码NG放料位[A]
AND P_1s
OR 851.09  ; 进料伺服Z轴#2夹爪扫码NG放料位标志
OUT 951.09  ; 进料伺服Z轴#2夹爪扫码NG放料位[lamp]
; rung 29
LD 451.10  ; 进料伺服Z轴#1夹爪配对取放料位[M]
OR 651.10  ; 进料伺服Z轴#1夹爪配对取放料位[A]
AND P_1s
OR 851.10  ; 进料伺服Z轴#1夹爪配对取放料位标志
OUT 951.10  ; 进料伺服Z轴#1夹爪配对取放料位[lamp]
; rung 30
LD 451.11  ; 进料伺服Z轴#2夹爪配对取放料位[M]
OR 651.11  ; 进料伺服Z轴#2夹爪配对取放料位[A]
AND P_1s
OR 851.11  ; 进料伺服Z轴#2夹爪配对取放料位标志
OUT 951.11  ; 进料伺服Z轴#2夹爪配对取放料位[lamp]

### Section 外部输出

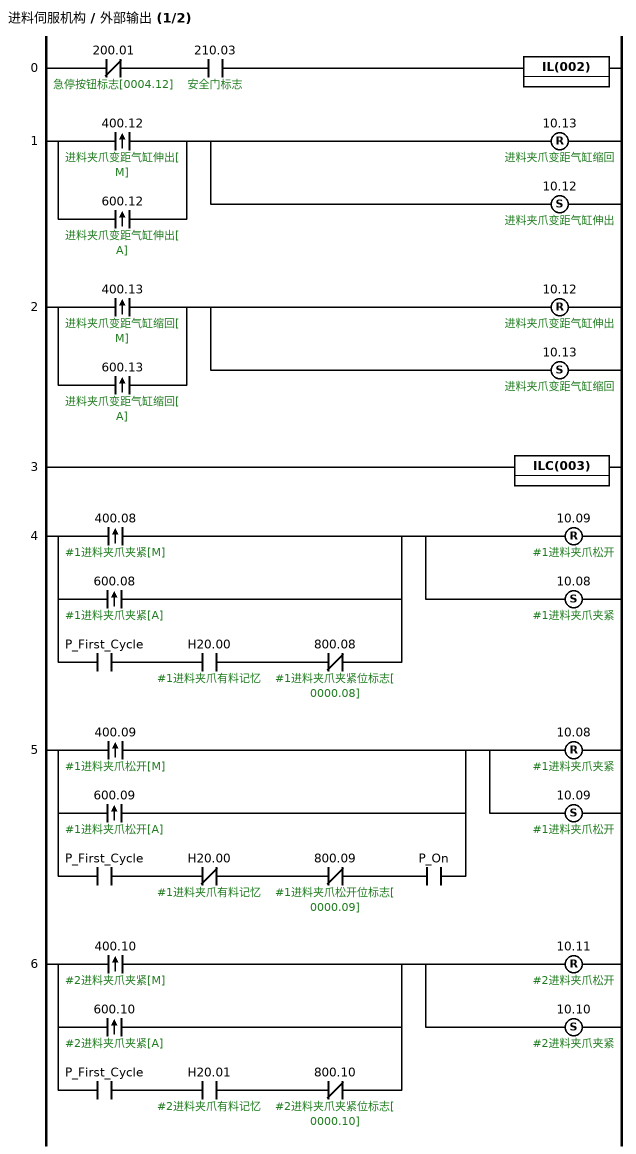
; rung 0
LDNOT 200.01  ; 急停按钮标志[0004.12]
AND 210.03  ; 安全门标志
IL(002)
; rung 1
@LD 400.12  ; 进料夹爪变距气缸伸出[M]
@OR 600.12  ; 进料夹爪变距气缸伸出[A]
RSET 10.13  ; 进料夹爪变距气缸缩回
SET 10.12  ; 进料夹爪变距气缸伸出
; rung 2
@LD 400.13  ; 进料夹爪变距气缸缩回[M]
@OR 600.13  ; 进料夹爪变距气缸缩回[A]
RSET 10.12  ; 进料夹爪变距气缸伸出
SET 10.13  ; 进料夹爪变距气缸缩回
; rung 3
ILC(003)
; rung 4
@LD 400.08  ; #1进料夹爪夹紧[M]
@OR 600.08  ; #1进料夹爪夹紧[A]
LD P_First_Cycle
AND H20.00  ; #1进料夹爪有料记忆
ANDNOT 800.08  ; #1进料夹爪夹紧位标志[0000.08]
ORLD
RSET 10.09  ; #1进料夹爪松开
SET 10.08  ; #1进料夹爪夹紧
; rung 5
@LD 400.09  ; #1进料夹爪松开[M]
@OR 600.09  ; #1进料夹爪松开[A]
LD P_First_Cycle
ANDNOT H20.00  ; #1进料夹爪有料记忆
ANDNOT 800.09  ; #1进料夹爪松开位标志[0000.09]
AND P_On
ORLD
RSET 10.08  ; #1进料夹爪夹紧
SET 10.09  ; #1进料夹爪松开
; rung 6
@LD 400.10  ; #2进料夹爪夹紧[M]
@OR 600.10  ; #2进料夹爪夹紧[A]
LD P_First_Cycle
AND H20.01  ; #2进料夹爪有料记忆
ANDNOT 800.10  ; #2进料夹爪夹紧位标志[0000.10]
ORLD
RSET 10.11  ; #2进料夹爪松开
SET 10.10  ; #2进料夹爪夹紧

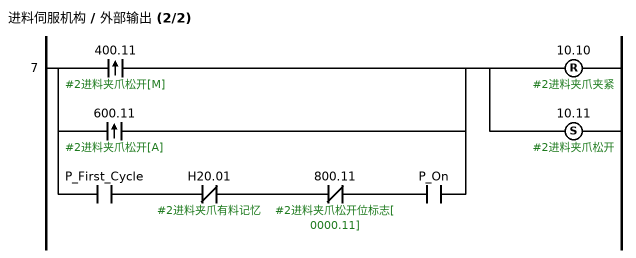
; rung 7
@LD 400.11  ; #2进料夹爪松开[M]
@OR 600.11  ; #2进料夹爪松开[A]
LD P_First_Cycle
ANDNOT H20.01  ; #2进料夹爪有料记忆
ANDNOT 800.11  ; #2进料夹爪松开位标志[0000.11]
AND P_On
ORLD
RSET 10.10  ; #2进料夹爪夹紧
SET 10.11  ; #2进料夹爪松开

### Section END
; rung 0
END(001)

## Program 氦检机构 (cyclic task 3)
Local symbols
up BOOL

### Section Main

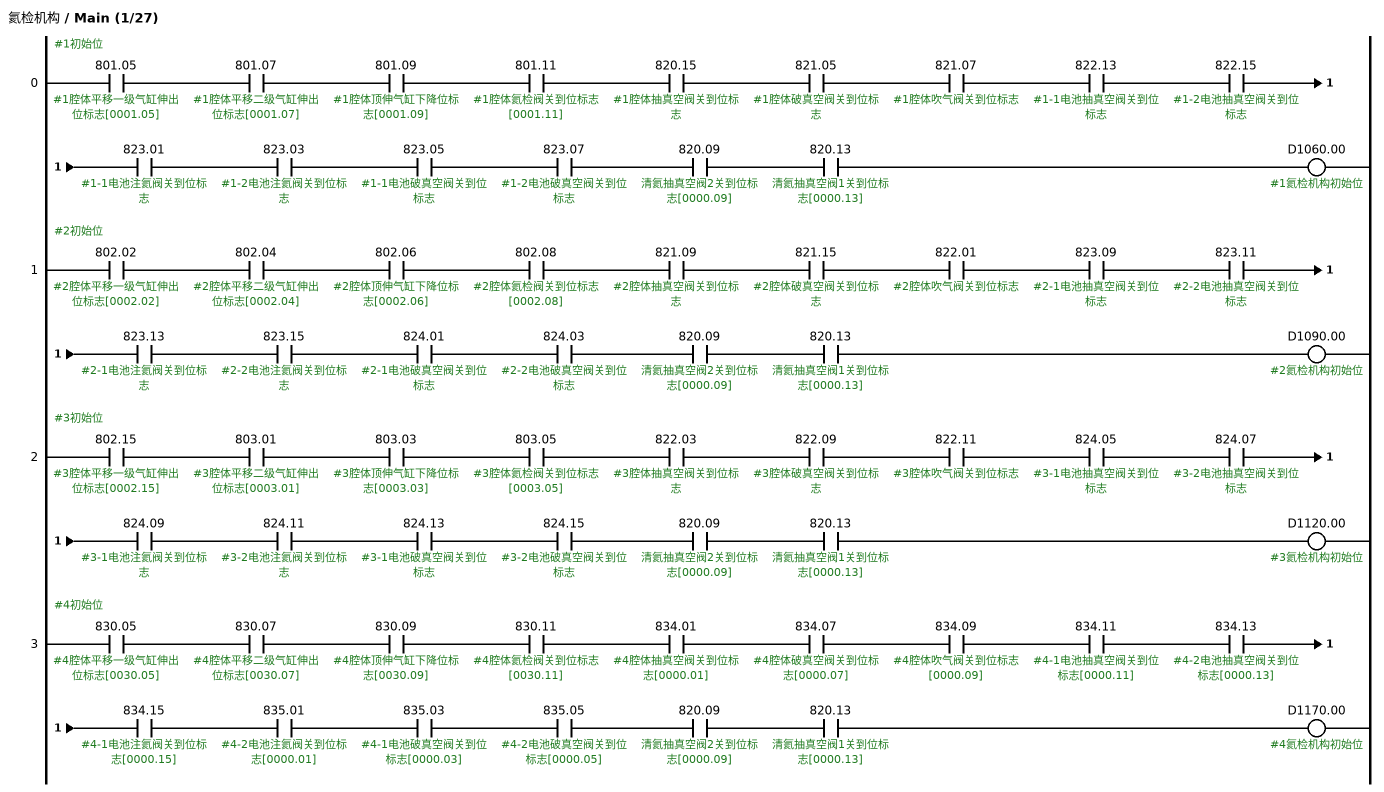
; rung 0: #1初始位
LD 801.05  ; #1腔体平移一级气缸伸出位标志[0001.05]
AND 801.07  ; #1腔体平移二级气缸伸出位标志[0001.07]
AND 801.09  ; #1腔体顶伸气缸下降位标志[0001.09]
AND 801.11  ; #1腔体氦检阀关到位标志[0001.11]
AND 820.15  ; #1腔体抽真空阀关到位标志
AND 821.05  ; #1腔体破真空阀关到位标志
AND 821.07  ; #1腔体吹气阀关到位标志
AND 822.13  ; #1-1电池抽真空阀关到位标志
AND 822.15  ; #1-2电池抽真空阀关到位标志
AND 823.01  ; #1-1电池注氦阀关到位标志
AND 823.03  ; #1-2电池注氦阀关到位标志
AND 823.05  ; #1-1电池破真空阀关到位标志
AND 823.07  ; #1-2电池破真空阀关到位标志
AND 820.09  ; 清氦抽真空阀2关到位标志[0000.09]
AND 820.13  ; 清氦抽真空阀1关到位标志[0000.13]
OUT D1060.00  ; #1氦检机构初始位
; rung 1: #2初始位
LD 802.02  ; #2腔体平移一级气缸伸出位标志[0002.02]
AND 802.04  ; #2腔体平移二级气缸伸出位标志[0002.04]
AND 802.06  ; #2腔体顶伸气缸下降位标志[0002.06]
AND 802.08  ; #2腔体氦检阀关到位标志[0002.08]
AND 821.09  ; #2腔体抽真空阀关到位标志
AND 821.15  ; #2腔体破真空阀关到位标志
AND 822.01  ; #2腔体吹气阀关到位标志
AND 823.09  ; #2-1电池抽真空阀关到位标志
AND 823.11  ; #2-2电池抽真空阀关到位标志
AND 823.13  ; #2-1电池注氦阀关到位标志
AND 823.15  ; #2-2电池注氦阀关到位标志
AND 824.01  ; #2-1电池破真空阀关到位标志
AND 824.03  ; #2-2电池破真空阀关到位标志
AND 820.09  ; 清氦抽真空阀2关到位标志[0000.09]
AND 820.13  ; 清氦抽真空阀1关到位标志[0000.13]
OUT D1090.00  ; #2氦检机构初始位
; rung 2: #3初始位
LD 802.15  ; #3腔体平移一级气缸伸出位标志[0002.15]
AND 803.01  ; #3腔体平移二级气缸伸出位标志[0003.01]
AND 803.03  ; #3腔体顶伸气缸下降位标志[0003.03]
AND 803.05  ; #3腔体氦检阀关到位标志[0003.05]
AND 822.03  ; #3腔体抽真空阀关到位标志
AND 822.09  ; #3腔体破真空阀关到位标志
AND 822.11  ; #3腔体吹气阀关到位标志
AND 824.05  ; #3-1电池抽真空阀关到位标志
AND 824.07  ; #3-2电池抽真空阀关到位标志
AND 824.09  ; #3-1电池注氦阀关到位标志
AND 824.11  ; #3-2电池注氦阀关到位标志
AND 824.13  ; #3-1电池破真空阀关到位标志
AND 824.15  ; #3-2电池破真空阀关到位标志
AND 820.09  ; 清氦抽真空阀2关到位标志[0000.09]
AND 820.13  ; 清氦抽真空阀1关到位标志[0000.13]
OUT D1120.00  ; #3氦检机构初始位
; rung 3: #4初始位
LD 830.05  ; #4腔体平移一级气缸伸出位标志[0030.05]
AND 830.07  ; #4腔体平移二级气缸伸出位标志[0030.07]
AND 830.09  ; #4腔体顶伸气缸下降位标志[0030.09]
AND 830.11  ; #4腔体氦检阀关到位标志[0030.11]
AND 834.01  ; #4腔体抽真空阀关到位标志[0000.01]
AND 834.07  ; #4腔体破真空阀关到位标志[0000.07]
AND 834.09  ; #4腔体吹气阀关到位标志[0000.09]
AND 834.11  ; #4-1电池抽真空阀关到位标志[0000.11]
AND 834.13  ; #4-2电池抽真空阀关到位标志[0000.13]
AND 834.15  ; #4-1电池注氦阀关到位标志[0000.15]
AND 835.01  ; #4-2电池注氦阀关到位标志[0000.01]
AND 835.03  ; #4-1电池破真空阀关到位标志[0000.03]
AND 835.05  ; #4-2电池破真空阀关到位标志[0000.05]
AND 820.09  ; 清氦抽真空阀2关到位标志[0000.09]
AND 820.13  ; 清氦抽真空阀1关到位标志[0000.13]
OUT D1170.00  ; #4氦检机构初始位

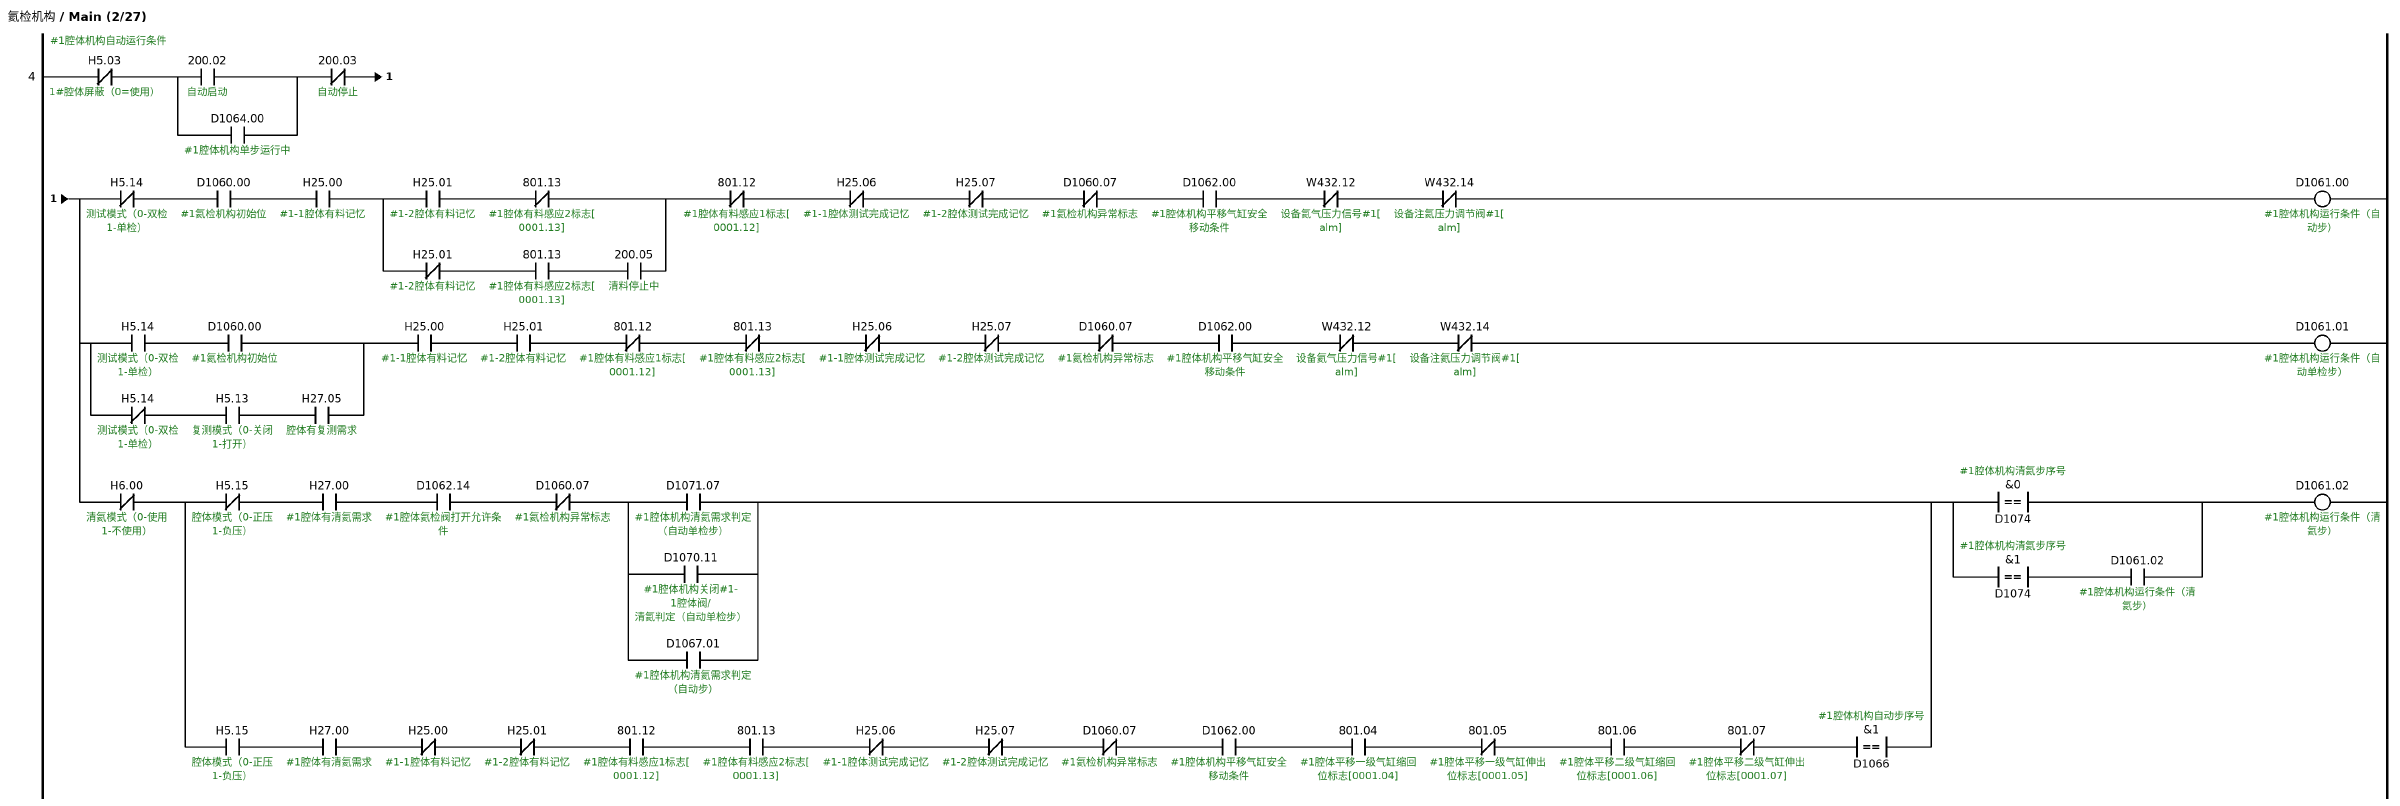
; rung 4: #1腔体机构自动运行条件
LDNOT H5.03  ; 1#腔体屏蔽（0=使用）
LD 200.02  ; 自动启动
OR D1064.00  ; #1腔体机构单步运行中
ANDLD
ANDNOT 200.03  ; 自动停止
OUT TR0
ANDNOT H5.14  ; 测试模式（0-双检 1-单检）
AND D1060.00  ; #1氦检机构初始位
AND H25.00  ; #1-1腔体有料记忆
LD H25.01  ; #1-2腔体有料记忆
ANDNOT 801.13  ; #1腔体有料感应2标志[0001.13]
LDNOT H25.01  ; #1-2腔体有料记忆
AND 801.13  ; #1腔体有料感应2标志[0001.13]
AND 200.05  ; 清料停止中
ORLD
ANDLD
ANDNOT 801.12  ; #1腔体有料感应1标志[0001.12]
ANDNOT H25.06  ; #1-1腔体测试完成记忆
ANDNOT H25.07  ; #1-2腔体测试完成记忆
ANDNOT D1060.07  ; #1氦检机构异常标志
AND D1062.00  ; #1腔体机构平移气缸安全移动条件
ANDNOT W432.12  ; 设备氦气压力信号#1[alm]
ANDNOT W432.14  ; 设备注氦压力调节阀#1[alm]
OUT D1061.00  ; #1腔体机构运行条件（自动步）
LD TR0
LD H5.14  ; 测试模式（0-双检 1-单检）
AND D1060.00  ; #1氦检机构初始位
LDNOT H5.14  ; 测试模式（0-双检 1-单检）
AND H5.13  ; 复测模式（0-关闭 1-打开）
AND H27.05  ; 腔体有复测需求
ORLD
ANDLD
AND H25.00  ; #1-1腔体有料记忆
AND H25.01  ; #1-2腔体有料记忆
ANDNOT 801.12  ; #1腔体有料感应1标志[0001.12]
ANDNOT 801.13  ; #1腔体有料感应2标志[0001.13]
ANDNOT H25.06  ; #1-1腔体测试完成记忆
ANDNOT H25.07  ; #1-2腔体测试完成记忆
ANDNOT D1060.07  ; #1氦检机构异常标志
AND D1062.00  ; #1腔体机构平移气缸安全移动条件
ANDNOT W432.12  ; 设备氦气压力信号#1[alm]
ANDNOT W432.14  ; 设备注氦压力调节阀#1[alm]
OUT D1061.01  ; #1腔体机构运行条件（自动单检步）
LD TR0
ANDNOT H6.00  ; 清氦模式（0-使用 1-不使用）
LDNOT H5.15  ; 腔体模式（0-正压 1-负压）
AND H27.00  ; #1腔体有清氦需求
AND D1062.14  ; #1腔体氦检阀打开允许条件
ANDNOT D1060.07  ; #1氦检机构异常标志
LD D1071.07  ; #1腔体机构清氦需求判定（自动单检步）
OR D1070.11  ; #1腔体机构关闭#1-1腔体阀/清氦判定（自动单检步）
OR D1067.01  ; #1腔体机构清氦需求判定（自动步）
ANDLD
LD H5.15  ; 腔体模式（0-正压 1-负压）
AND H27.00  ; #1腔体有清氦需求
ANDNOT H25.00  ; #1-1腔体有料记忆
ANDNOT H25.01  ; #1-2腔体有料记忆
AND 801.12  ; #1腔体有料感应1标志[0001.12]
AND 801.13  ; #1腔体有料感应2标志[0001.13]
ANDNOT H25.06  ; #1-1腔体测试完成记忆
ANDNOT H25.07  ; #1-2腔体测试完成记忆
ANDNOT D1060.07  ; #1氦检机构异常标志
AND D1062.00  ; #1腔体机构平移气缸安全移动条件
AND 801.04  ; #1腔体平移一级气缸缩回位标志[0001.04]
ANDNOT 801.05  ; #1腔体平移一级气缸伸出位标志[0001.05]
AND 801.06  ; #1腔体平移二级气缸缩回位标志[0001.06]
ANDNOT 801.07  ; #1腔体平移二级气缸伸出位标志[0001.07]
AND=L(301) &1 D1066  ; #1腔体机构自动步序号
ORLD
ANDLD
LD=L(301) &0 D1074  ; #1腔体机构清氦步序号
LD=L(301) &1 D1074  ; #1腔体机构清氦步序号
AND D1061.02  ; #1腔体机构运行条件（清氦步）
ORLD
ANDLD
OUT D1061.02  ; #1腔体机构运行条件（清氦步）

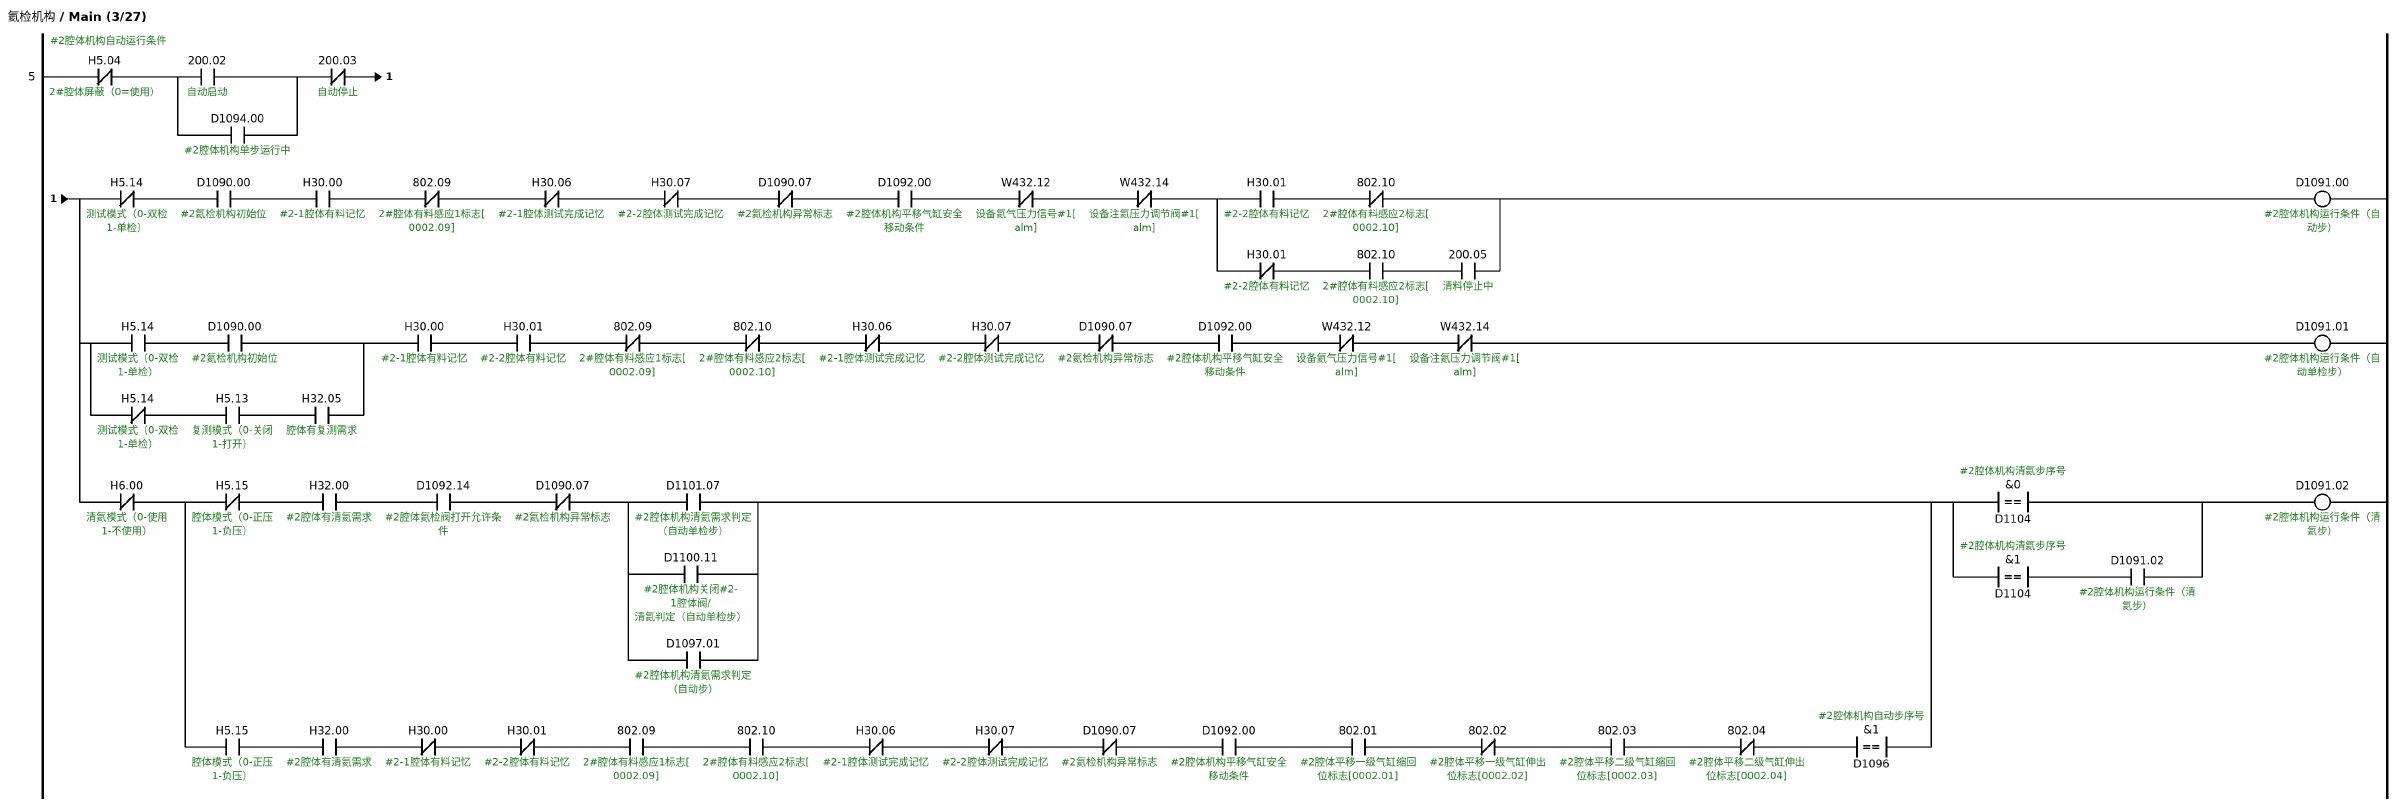
; rung 5: #2腔体机构自动运行条件
LDNOT H5.04  ; 2#腔体屏蔽（0=使用）
LD 200.02  ; 自动启动
OR D1094.00  ; #2腔体机构单步运行中
ANDLD
ANDNOT 200.03  ; 自动停止
OUT TR0
ANDNOT H5.14  ; 测试模式（0-双检 1-单检）
AND D1090.00  ; #2氦检机构初始位
AND H30.00  ; #2-1腔体有料记忆
ANDNOT 802.09  ; 2#腔体有料感应1标志[0002.09]
ANDNOT H30.06  ; #2-1腔体测试完成记忆
ANDNOT H30.07  ; #2-2腔体测试完成记忆
ANDNOT D1090.07  ; #2氦检机构异常标志
AND D1092.00  ; #2腔体机构平移气缸安全移动条件
ANDNOT W432.12  ; 设备氦气压力信号#1[alm]
ANDNOT W432.14  ; 设备注氦压力调节阀#1[alm]
LD H30.01  ; #2-2腔体有料记忆
ANDNOT 802.10  ; 2#腔体有料感应2标志[0002.10]
LDNOT H30.01  ; #2-2腔体有料记忆
AND 802.10  ; 2#腔体有料感应2标志[0002.10]
AND 200.05  ; 清料停止中
ORLD
ANDLD
OUT D1091.00  ; #2腔体机构运行条件（自动步）
LD TR0
LD H5.14  ; 测试模式（0-双检 1-单检）
AND D1090.00  ; #2氦检机构初始位
LDNOT H5.14  ; 测试模式（0-双检 1-单检）
AND H5.13  ; 复测模式（0-关闭 1-打开）
AND H32.05  ; 腔体有复测需求
ORLD
ANDLD
AND H30.00  ; #2-1腔体有料记忆
AND H30.01  ; #2-2腔体有料记忆
ANDNOT 802.09  ; 2#腔体有料感应1标志[0002.09]
ANDNOT 802.10  ; 2#腔体有料感应2标志[0002.10]
ANDNOT H30.06  ; #2-1腔体测试完成记忆
ANDNOT H30.07  ; #2-2腔体测试完成记忆
ANDNOT D1090.07  ; #2氦检机构异常标志
AND D1092.00  ; #2腔体机构平移气缸安全移动条件
ANDNOT W432.12  ; 设备氦气压力信号#1[alm]
ANDNOT W432.14  ; 设备注氦压力调节阀#1[alm]
OUT D1091.01  ; #2腔体机构运行条件（自动单检步）
LD TR0
ANDNOT H6.00  ; 清氦模式（0-使用 1-不使用）
LDNOT H5.15  ; 腔体模式（0-正压 1-负压）
AND H32.00  ; #2腔体有清氦需求
AND D1092.14  ; #2腔体氦检阀打开允许条件
ANDNOT D1090.07  ; #2氦检机构异常标志
LD D1101.07  ; #2腔体机构清氦需求判定（自动单检步）
OR D1100.11  ; #2腔体机构关闭#2-1腔体阀/清氦判定（自动单检步）
OR D1097.01  ; #2腔体机构清氦需求判定（自动步）
ANDLD
LD H5.15  ; 腔体模式（0-正压 1-负压）
AND H32.00  ; #2腔体有清氦需求
ANDNOT H30.00  ; #2-1腔体有料记忆
ANDNOT H30.01  ; #2-2腔体有料记忆
AND 802.09  ; 2#腔体有料感应1标志[0002.09]
AND 802.10  ; 2#腔体有料感应2标志[0002.10]
ANDNOT H30.06  ; #2-1腔体测试完成记忆
ANDNOT H30.07  ; #2-2腔体测试完成记忆
ANDNOT D1090.07  ; #2氦检机构异常标志
AND D1092.00  ; #2腔体机构平移气缸安全移动条件
AND 802.01  ; #2腔体平移一级气缸缩回位标志[0002.01]
ANDNOT 802.02  ; #2腔体平移一级气缸伸出位标志[0002.02]
AND 802.03  ; #2腔体平移二级气缸缩回位标志[0002.03]
ANDNOT 802.04  ; #2腔体平移二级气缸伸出位标志[0002.04]
AND=L(301) &1 D1096  ; #2腔体机构自动步序号
ORLD
ANDLD
LD=L(301) &0 D1104  ; #2腔体机构清氦步序号
LD=L(301) &1 D1104  ; #2腔体机构清氦步序号
AND D1091.02  ; #2腔体机构运行条件（清氦步）
ORLD
ANDLD
OUT D1091.02  ; #2腔体机构运行条件（清氦步）

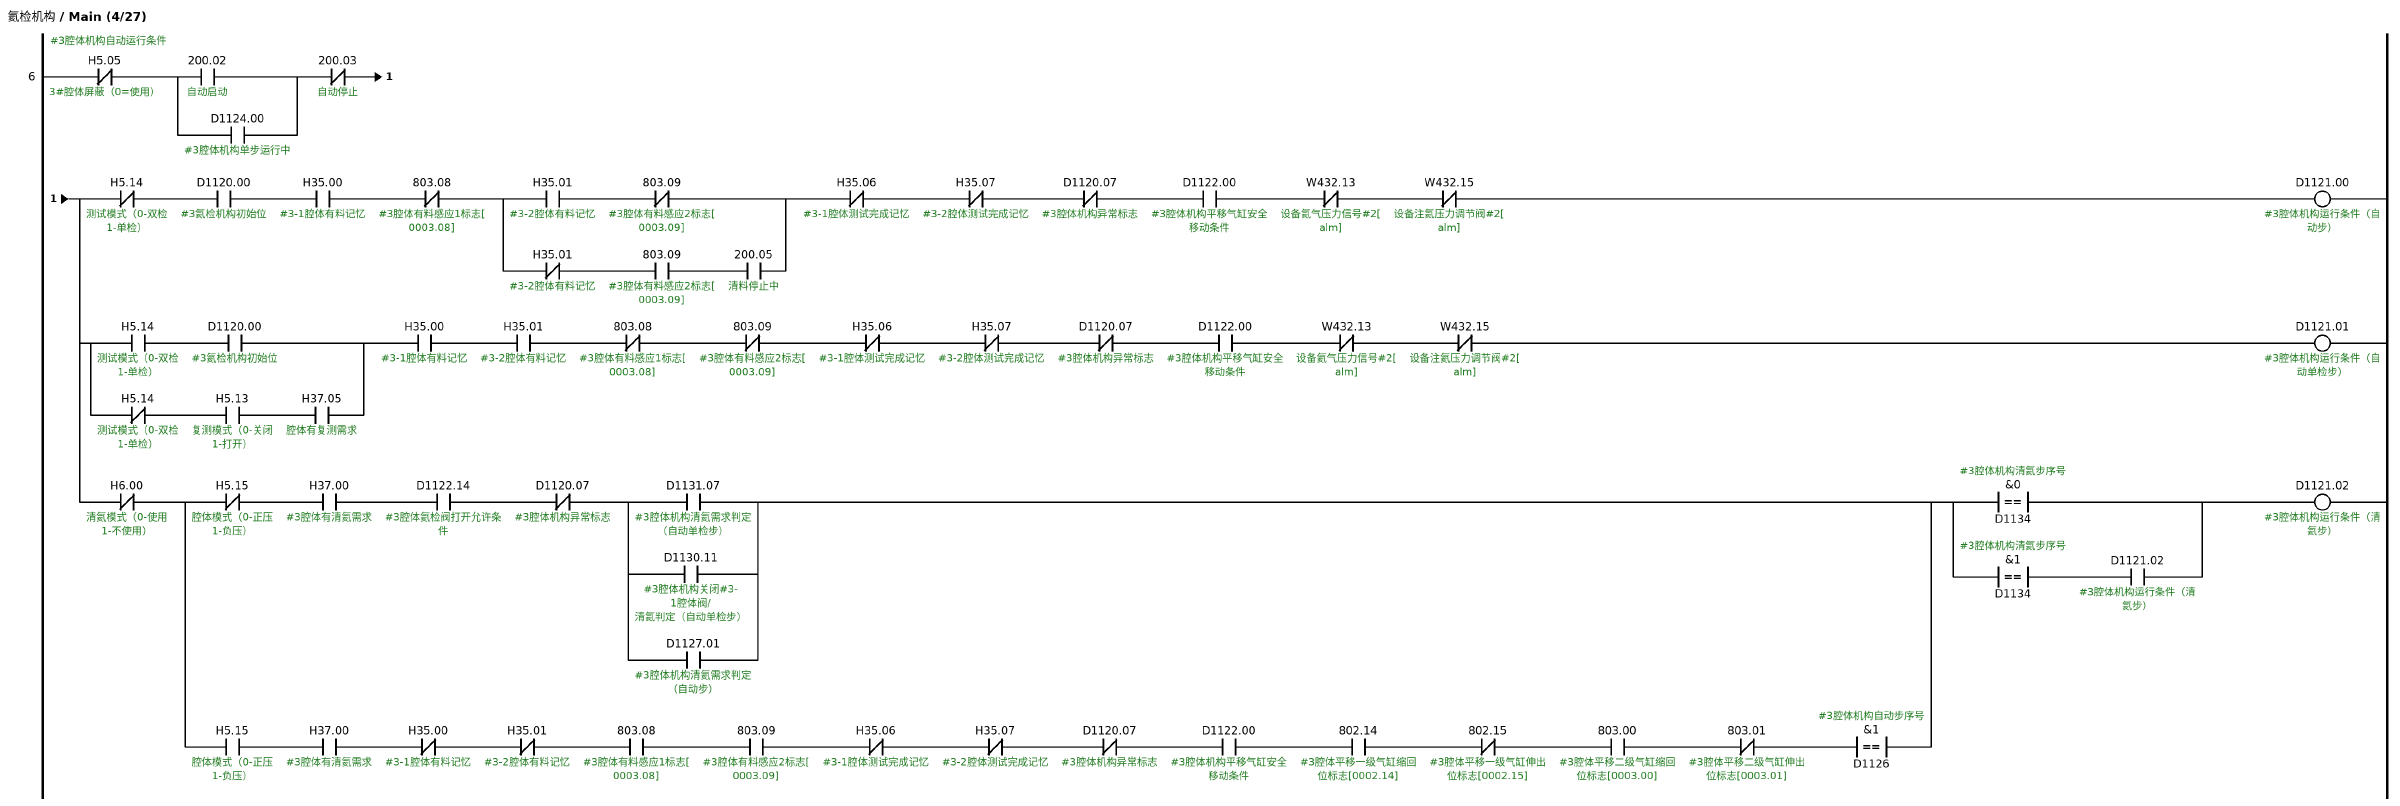
; rung 6: #3腔体机构自动运行条件
LDNOT H5.05  ; 3#腔体屏蔽（0=使用）
LD 200.02  ; 自动启动
OR D1124.00  ; #3腔体机构单步运行中
ANDLD
ANDNOT 200.03  ; 自动停止
OUT TR0
ANDNOT H5.14  ; 测试模式（0-双检 1-单检）
AND D1120.00  ; #3氦检机构初始位
AND H35.00  ; #3-1腔体有料记忆
ANDNOT 803.08  ; #3腔体有料感应1标志[0003.08]
LD H35.01  ; #3-2腔体有料记忆
ANDNOT 803.09  ; #3腔体有料感应2标志[0003.09]
LDNOT H35.01  ; #3-2腔体有料记忆
AND 803.09  ; #3腔体有料感应2标志[0003.09]
AND 200.05  ; 清料停止中
ORLD
ANDLD
ANDNOT H35.06  ; #3-1腔体测试完成记忆
ANDNOT H35.07  ; #3-2腔体测试完成记忆
ANDNOT D1120.07  ; #3腔体机构异常标志
AND D1122.00  ; #3腔体机构平移气缸安全移动条件
ANDNOT W432.13  ; 设备氦气压力信号#2[alm]
ANDNOT W432.15  ; 设备注氦压力调节阀#2[alm]
OUT D1121.00  ; #3腔体机构运行条件（自动步）
LD TR0
LD H5.14  ; 测试模式（0-双检 1-单检）
AND D1120.00  ; #3氦检机构初始位
LDNOT H5.14  ; 测试模式（0-双检 1-单检）
AND H5.13  ; 复测模式（0-关闭 1-打开）
AND H37.05  ; 腔体有复测需求
ORLD
ANDLD
AND H35.00  ; #3-1腔体有料记忆
AND H35.01  ; #3-2腔体有料记忆
ANDNOT 803.08  ; #3腔体有料感应1标志[0003.08]
ANDNOT 803.09  ; #3腔体有料感应2标志[0003.09]
ANDNOT H35.06  ; #3-1腔体测试完成记忆
ANDNOT H35.07  ; #3-2腔体测试完成记忆
ANDNOT D1120.07  ; #3腔体机构异常标志
AND D1122.00  ; #3腔体机构平移气缸安全移动条件
ANDNOT W432.13  ; 设备氦气压力信号#2[alm]
ANDNOT W432.15  ; 设备注氦压力调节阀#2[alm]
OUT D1121.01  ; #3腔体机构运行条件（自动单检步）
LD TR0
ANDNOT H6.00  ; 清氦模式（0-使用 1-不使用）
LDNOT H5.15  ; 腔体模式（0-正压 1-负压）
AND H37.00  ; #3腔体有清氦需求
AND D1122.14  ; #3腔体氦检阀打开允许条件
ANDNOT D1120.07  ; #3腔体机构异常标志
LD D1131.07  ; #3腔体机构清氦需求判定（自动单检步）
OR D1130.11  ; #3腔体机构关闭#3-1腔体阀/清氦判定（自动单检步）
OR D1127.01  ; #3腔体机构清氦需求判定（自动步）
ANDLD
LD H5.15  ; 腔体模式（0-正压 1-负压）
AND H37.00  ; #3腔体有清氦需求
ANDNOT H35.00  ; #3-1腔体有料记忆
ANDNOT H35.01  ; #3-2腔体有料记忆
AND 803.08  ; #3腔体有料感应1标志[0003.08]
AND 803.09  ; #3腔体有料感应2标志[0003.09]
ANDNOT H35.06  ; #3-1腔体测试完成记忆
ANDNOT H35.07  ; #3-2腔体测试完成记忆
ANDNOT D1120.07  ; #3腔体机构异常标志
AND D1122.00  ; #3腔体机构平移气缸安全移动条件
AND 802.14  ; #3腔体平移一级气缸缩回位标志[0002.14]
ANDNOT 802.15  ; #3腔体平移一级气缸伸出位标志[0002.15]
AND 803.00  ; #3腔体平移二级气缸缩回位标志[0003.00]
ANDNOT 803.01  ; #3腔体平移二级气缸伸出位标志[0003.01]
AND=L(301) &1 D1126  ; #3腔体机构自动步序号
ORLD
ANDLD
LD=L(301) &0 D1134  ; #3腔体机构清氦步序号
LD=L(301) &1 D1134  ; #3腔体机构清氦步序号
AND D1121.02  ; #3腔体机构运行条件（清氦步）
ORLD
ANDLD
OUT D1121.02  ; #3腔体机构运行条件（清氦步）

